LIN {X 0,Y 536.423,Z 174.915,A -85,B 0,C 180,E1 25056.548,E2 25056.548} C_VEL
LIN {X 0,Y 536.456,Z 174.916,A -85,B 0,C 180,E1 25053.19,E2 25053.19} C_VEL
LIN {X 0,Y 536.429,Z 174.979,A -85,B 0,C 180,E1 25052.229,E2 25052.229} C_VEL
LIN {X 0,Y 538.274,Z 182.198,A -85,B 0,C 180,E1 25051.657,E2 25051.657} C_VEL
LIN {X 0,Y 539.189,Z 215.155,A -85,B 0,C 180,E1 25049.25,E2 25049.25} C_VEL
LIN {X 0,Y 539.582,Z 245.329,A -85,B 0,C 180,E1 25046.881,E2 25046.881} C_VEL
LIN {X 0,Y 539.681,Z 277.796,A -85,B 0,C 180,E1 25044.228,E2 25044.228} C_VEL
LIN {X 0,Y 539.301,Z 312.385,A -85,B 0,C 180,E1 25041.251,E2 25041.251} C_VEL
LIN {X 0,Y 539.248,Z 319.143,A -85,B 0,C 180,E1 25040.702,E2 25040.702} C_VEL
LIN {X 0,Y 539.576,Z 325.813,A -85,B 0,C 180,E1 25040.595,E2 25040.595} C_VEL
LIN {X 0,Y 538.831,Z 486.501,A -85,B 0,C 180,E1 25038.368,E2 25038.368} C_VEL
LIN {X 0,Y 538.703,Z 503.712,A -85,B 0,C 180,E1 25037.931,E2 25037.931} C_VEL
LIN {X 0,Y 538.465,Z 519.532,A -85,B 0,C 180,E1 25037.339,E2 25037.339} C_VEL
LIN {X 0,Y 538.129,Z 535.901,A -85,B 0,C 180,E1 25036.514,E2 25036.514} C_VEL
LIN {X 0,Y 537.753,Z 551.043,A -85,B 0,C 180,E1 25035.53,E2 25035.53} C_VEL
LIN {X 0,Y 537.349,Z 564.974,A -85,B 0,C 180,E1 25034.383,E2 25034.383} C_VEL
LIN {X 0,Y 536.941,Z 578.306,A -85,B 0,C 180,E1 25033.021,E2 25033.021} C_VEL
LIN {X 0,Y 536.586,Z 589.487,A -85,B 0,C 180,E1 25031.609,E2 25031.609} C_VEL
LIN {X 0,Y 536.286,Z 599.811,A -85,B 0,C 180,E1 25029.985,E2 25029.985} C_VEL
LIN {X 0,Y 536.079,Z 608.451,A -85,B 0,C 180,E1 25028.257,E2 25028.257} C_VEL
LIN {X 0,Y 535.975,Z 615.684,A -85,B 0,C 180,E1 25026.426,E2 25026.426} C_VEL
LIN {X 0,Y 535.936,Z 620.745,A -85,B 0,C 180,E1 25024.708,E2 25024.708} C_VEL
LIN {X 0,Y 535.917,Z 624.48,A -85,B 0,C 180,E1 25022.78,E2 25022.78} C_VEL
LIN {X 0,Y 535.91,Z 626.276,A -85,B 0,C 180,E1 25020.855,E2 25020.855} C_VEL
LIN {X 0,Y 535.911,Z 626.268,A -85,B 0,C 180,E1 25019.038,E2 25019.038} C_VEL
LIN {X 0,Y 535.913,Z 624.459,A -85,B 0,C 180,E1 25017.112,E2 25017.112} C_VEL
LIN {X 0,Y 535.931,Z 620.697,A -85,B 0,C 180,E1 25015.184,E2 25015.184} C_VEL
LIN {X 0,Y 535.979,Z 615.244,A -85,B 0,C 180,E1 25013.358,E2 25013.358} C_VEL
LIN {X 0,Y 536.088,Z 607.834,A -85,B 0,C 180,E1 25011.527,E2 25011.527} C_VEL
LIN {X 0,Y 536.285,Z 599.404,A -85,B 0,C 180,E1 25009.872,E2 25009.872} C_VEL
LIN {X 0,Y 536.566,Z 589.166,A -85,B 0,C 180,E1 25008.28,E2 25008.28} C_VEL
LIN {X 0,Y 536.909,Z 577.887,A -85,B 0,C 180,E1 25006.868,E2 25006.868} C_VEL
LIN {X 0,Y 537.301,Z 565.067,A -85,B 0,C 180,E1 25005.56,E2 25005.56} C_VEL
LIN {X 0,Y 537.724,Z 550.492,A -85,B 0,C 180,E1 25004.358,E2 25004.358} C_VEL
LIN {X 0,Y 538.125,Z 535.397,A -85,B 0,C 180,E1 25003.373,E2 25003.373} C_VEL
LIN {X 0,Y 538.466,Z 519.15,A -85,B 0,C 180,E1 25002.549,E2 25002.549} C_VEL
LIN {X 0,Y 538.78,Z 502.032,A -85,B 0,C 180,E1 25001.907,E2 25001.907} C_VEL
LIN {X 0,Y 538.968,Z 484.452,A -85,B 0,C 180,E1 25001.468,E2 25001.468} C_VEL
LIN {X 0,Y 539.448,Z 388.201,A -85,B 0,C 180,E1 25000.124,E2 25000.124} C_VEL
LIN {X 0,Y 538.575,Z 380.596,A -85,B 0,C 180,E1 24999.986,E2 24999.986} C_VEL
LIN {X 0,Y 532.766,Z 360.688,A -85,B 0,C 180,E1 24999.487,E2 24999.487} C_VEL
LIN {X 0,Y 532.096,Z 354.154,A -85,B 0,C 180,E1 24999.367,E2 24999.367} C_VEL
LIN {X 0,Y 532.09,Z 321.506,A -85,B 0,C 180,E1 24998.896,E2 24998.896} C_VEL
LIN {X 0,Y 531.331,Z 316.809,A -85,B 0,C 180,E1 24998.79,E2 24998.79} C_VEL
LIN {X 0,Y 532.06,Z 279.719,A -85,B 0,C 180,E1 24995.408,E2 24995.408} C_VEL
LIN {X 0,Y 532.553,Z 244.005,A -85,B 0,C 180,E1 24992.165,E2 24992.165} C_VEL
LIN {X 0,Y 532.935,Z 207.634,A -85,B 0,C 180,E1 24988.87,E2 24988.87} C_VEL
LIN {X 0,Y 533.056,Z 191.079,A -85,B 0,C 180,E1 24987.373,E2 24987.373} C_VEL
LIN {X 0,Y 528.507,Z 175.902,A -85,B 0,C 180,E1 24985.715,E2 24985.715} C_VEL
LIN {X 0,Y 528.552,Z 176.121,A -85,B 0,C 180,E1 24984.625,E2 24984.625} C_VEL
LIN {X 0,Y 529.932,Z 179.548,A -85,B 0,C 180,E1 24984.453,E2 24984.453} C_VEL
LIN {X 0,Y 531.563,Z 181.867,A -85,B 0,C 180,E1 24984.281,E2 24984.281} C_VEL
LIN {X 0,Y 541.38,Z 197.994,A -85,B 0,C 180,E1 24983.233,E2 24983.233} C_VEL
LIN {X 0,Y 539.048,Z 419.645,A -85,B 0,C 180,E1 24979.896,E2 24979.896} C_VEL
LIN {X 0,Y 538.527,Z 464.266,A -85,B 0,C 180,E1 24979.196,E2 24979.196} C_VEL
LIN {X 0,Y 537.87,Z 485.766,A -85,B 0,C 180,E1 24978.667,E2 24978.667} C_VEL
LIN {X 0,Y 537.128,Z 506.444,A -85,B 0,C 180,E1 24977.965,E2 24977.965} C_VEL
LIN {X 0,Y 536.288,Z 525.333,A -85,B 0,C 180,E1 24977.154,E2 24977.154} C_VEL
LIN {X 0,Y 535.271,Z 545.952,A -85,B 0,C 180,E1 24976.063,E2 24976.063} C_VEL
LIN {X 0,Y 534.249,Z 564.528,A -85,B 0,C 180,E1 24974.875,E2 24974.875} C_VEL
LIN {X 0,Y 533.163,Z 583.881,A -85,B 0,C 180,E1 24973.418,E2 24973.418} C_VEL
LIN {X 0,Y 532.132,Z 600.696,A -85,B 0,C 180,E1 24971.92,E2 24971.92} C_VEL
LIN {X 0,Y 531.203,Z 617.415,A -85,B 0,C 180,E1 24970.212,E2 24970.212} C_VEL
LIN {X 0,Y 530.324,Z 633.077,A -85,B 0,C 180,E1 24968.337,E2 24968.337} C_VEL
LIN {X 0,Y 529.625,Z 646.645,A -85,B 0,C 180,E1 24966.463,E2 24966.463} C_VEL
LIN {X 0,Y 529.002,Z 660.204,A -85,B 0,C 180,E1 24964.281,E2 24964.281} C_VEL
LIN {X 0,Y 528.567,Z 671.632,A -85,B 0,C 180,E1 24962.111,E2 24962.111} C_VEL
LIN {X 0,Y 528.249,Z 682.226,A -85,B 0,C 180,E1 24959.681,E2 24959.681} C_VEL
LIN {X 0,Y 528.072,Z 689.894,A -85,B 0,C 180,E1 24957.516,E2 24957.516} C_VEL
LIN {X 0,Y 527.973,Z 696.696,A -85,B 0,C 180,E1 24955.101,E2 24955.101} C_VEL
LIN {X 0,Y 527.924,Z 701.372,A -85,B 0,C 180,E1 24952.846,E2 24952.846} C_VEL
LIN {X 0,Y 527.907,Z 704.615,A -85,B 0,C 180,E1 24950.511,E2 24950.511} C_VEL
LIN {X 0,Y 527.91,Z 706.258,A -85,B 0,C 180,E1 24948.097,E2 24948.097} C_VEL
LIN {X 0,Y 527.916,Z 706.289,A -85,B 0,C 180,E1 24945.94,E2 24945.94} C_VEL
LIN {X 0,Y 527.916,Z 704.805,A -85,B 0,C 180,E1 24943.583,E2 24943.583} C_VEL
LIN {X 0,Y 527.929,Z 701.693,A -85,B 0,C 180,E1 24941.249,E2 24941.249} C_VEL
LIN {X 0,Y 527.966,Z 697.241,A -85,B 0,C 180,E1 24939.044,E2 24939.044} C_VEL
LIN {X 0,Y 528.066,Z 690.659,A -85,B 0,C 180,E1 24936.633,E2 24936.633} C_VEL
LIN {X 0,Y 528.231,Z 683.073,A -85,B 0,C 180,E1 24934.451,E2 24934.451} C_VEL
LIN {X 0,Y 528.516,Z 673.375,A -85,B 0,C 180,E1 24932.169,E2 24932.169} C_VEL
LIN {X 0,Y 528.93,Z 662.117,A -85,B 0,C 180,E1 24929.97,E2 24929.97} C_VEL
LIN {X 0,Y 529.513,Z 649.292,A -85,B 0,C 180,E1 24927.836,E2 24927.836} C_VEL
LIN {X 0,Y 530.185,Z 635.52,A -85,B 0,C 180,E1 24925.891,E2 24925.891} C_VEL
LIN {X 0,Y 531.061,Z 619.631,A -85,B 0,C 180,E1 24923.948,E2 24923.948} C_VEL
LIN {X 0,Y 532.034,Z 602.565,A -85,B 0,C 180,E1 24922.169,E2 24922.169} C_VEL
LIN {X 0,Y 533.029,Z 585.876,A -85,B 0,C 180,E1 24920.662,E2 24920.662} C_VEL
LIN {X 0,Y 534.148,Z 566.313,A -85,B 0,C 180,E1 24919.157,E2 24919.157} C_VEL
LIN {X 0,Y 535.213,Z 547.196,A -85,B 0,C 180,E1 24917.923,E2 24917.923} C_VEL
LIN {X 0,Y 536.252,Z 526.209,A -85,B 0,C 180,E1 24916.797,E2 24916.797} C_VEL
LIN {X 0,Y 537.065,Z 507.68,A -85,B 0,C 180,E1 24915.994,E2 24915.994} C_VEL
LIN {X 0,Y 537.857,Z 487.102,A -85,B 0,C 180,E1 24915.28,E2 24915.28} C_VEL
LIN {X 0,Y 538.479,Z 465.319,A -85,B 0,C 180,E1 24914.736,E2 24914.736} C_VEL
LIN {X 0,Y 538.951,Z 430.041,A -85,B 0,C 180,E1 24914.169,E2 24914.169} C_VEL
LIN {X 0,Y 541.072,Z 221.448,A -85,B 0,C 180,E1 24911.031,E2 24911.031} C_VEL
LIN {X 0,Y 541.252,Z 197.496,A -85,B 0,C 180,E1 24910.659,E2 24910.659} C_VEL
LIN {X 0,Y 530.508,Z 180.267,A -85,B 0,C 180,E1 24909.507,E2 24909.507} C_VEL
LIN {X 0,Y 528.744,Z 177.007,A -85,B 0,C 180,E1 24909.3,E2 24909.3} C_VEL
LIN {X 0,Y 528.527,Z 175.903,A -85,B 0,C 180,E1 24909.234,E2 24909.234} C_VEL
LIN {X 0,Y 528.523,Z 175.903,A -85,B 0,C 180,E1 24905.763,E2 24905.763} C_VEL
LIN {X 0,Y 528.525,Z 175.902,A -85,B 0,C 180,E1 24902.265,E2 24902.265} C_VEL
LIN {X 0,Y 528.529,Z 175.899,A -85,B 0,C 180,E1 24898.77,E2 24898.77} C_VEL
LIN {X 0,Y 528.467,Z 175.902,A -85,B 0,C 180,E1 24895.417,E2 24895.417} C_VEL
LIN {X 0,Y 528.468,Z 175.898,A -85,B 0,C 180,E1 24892.056,E2 24892.056} C_VEL
LIN {X 0,Y 528.527,Z 175.892,A -85,B 0,C 180,E1 24888.827,E2 24888.827} C_VEL
LIN {X 0,Y 528.521,Z 175.894,A -85,B 0,C 180,E1 24885.343,E2 24885.343} C_VEL
LIN {X 0,Y 528.523,Z 175.899,A -85,B 0,C 180,E1 24881.898,E2 24881.898} C_VEL
LIN {X 0,Y 528.528,Z 175.901,A -85,B 0,C 180,E1 24878.446,E2 24878.446} C_VEL
LIN {X 0,Y 528.482,Z 175.901,A -85,B 0,C 180,E1 24875.111,E2 24875.111} C_VEL
LIN {X 0,Y 528.463,Z 175.896,A -85,B 0,C 180,E1 24871.735,E2 24871.735} C_VEL
LIN {X 0,Y 528.503,Z 175.896,A -85,B 0,C 180,E1 24868.351,E2 24868.351} C_VEL
LIN {X 0,Y 528.522,Z 175.899,A -85,B 0,C 180,E1 24864.953,E2 24864.953} C_VEL
LIN {X 0,Y 528.509,Z 175.902,A -85,B 0,C 180,E1 24861.442,E2 24861.442} C_VEL
LIN {X 0,Y 528.519,Z 175.894,A -85,B 0,C 180,E1 24858.075,E2 24858.075} C_VEL
LIN {X 0,Y 528.513,Z 175.903,A -85,B 0,C 180,E1 24854.685,E2 24854.685} C_VEL
LIN {X 0,Y 528.47,Z 175.904,A -85,B 0,C 180,E1 24851.348,E2 24851.348} C_VEL
LIN {X 0,Y 528.485,Z 175.897,A -85,B 0,C 180,E1 24847.939,E2 24847.939} C_VEL
LIN {X 0,Y 528.522,Z 175.889,A -85,B 0,C 180,E1 24844.558,E2 24844.558} C_VEL
LIN {X 0,Y 528.507,Z 175.898,A -85,B 0,C 180,E1 24841.193,E2 24841.193} C_VEL
LIN {X 0,Y 528.505,Z 175.903,A -85,B 0,C 180,E1 24837.723,E2 24837.723} C_VEL
LIN {X 0,Y 528.521,Z 175.901,A -85,B 0,C 180,E1 24834.319,E2 24834.319} C_VEL
LIN {X 0,Y 528.482,Z 175.9,A -85,B 0,C 180,E1 24830.966,E2 24830.966} C_VEL
LIN {X 0,Y 528.485,Z 175.898,A -85,B 0,C 180,E1 24827.656,E2 24827.656} C_VEL
LIN {X 0,Y 528.52,Z 175.896,A -85,B 0,C 180,E1 24824.305,E2 24824.305} C_VEL
LIN {X 0,Y 528.508,Z 175.901,A -85,B 0,C 180,E1 24820.896,E2 24820.896} C_VEL
LIN {X 0,Y 528.498,Z 175.904,A -85,B 0,C 180,E1 24817.405,E2 24817.405} C_VEL
LIN {X 0,Y 528.514,Z 175.9,A -85,B 0,C 180,E1 24814.087,E2 24814.087} C_VEL
LIN {X 0,Y 528.498,Z 175.899,A -85,B 0,C 180,E1 24810.66,E2 24810.66} C_VEL
LIN {X 0,Y 528.551,Z 176.084,A -85,B 0,C 180,E1 24808.369,E2 24808.369} C_VEL
LIN {X 0,Y 529.95,Z 179.609,A -85,B 0,C 180,E1 24807.901,E2 24807.901} C_VEL
LIN {X 0,Y 536.933,Z 193.998,A -85,B 0,C 180,E1 24805.909,E2 24805.909} C_VEL
LIN {X 0,Y 542.938,Z 206.96,A -85,B 0,C 180,E1 24804.219,E2 24804.219} C_VEL
LIN {X 0,Y 541.161,Z 250.131,A -85,B 0,C 180,E1 24800.896,E2 24800.896} C_VEL
LIN {X 0,Y 540.404,Z 281.034,A -85,B 0,C 180,E1 24798.533,E2 24798.533} C_VEL
LIN {X 0,Y 541.806,Z 294.589,A -85,B 0,C 180,E1 24797.37,E2 24797.37} C_VEL
LIN {X 0,Y 544.881,Z 306.361,A -85,B 0,C 180,E1 24796.228,E2 24796.228} C_VEL
LIN {X 0,Y 549.168,Z 315.707,A -85,B 0,C 180,E1 24795.203,E2 24795.203} C_VEL
LIN {X 0,Y 555.008,Z 323.69,A -85,B 0,C 180,E1 24794.193,E2 24794.193} C_VEL
LIN {X 0,Y 561.764,Z 329.796,A -85,B 0,C 180,E1 24793.285,E2 24793.285} C_VEL
LIN {X 0,Y 569.988,Z 334.684,A -85,B 0,C 180,E1 24792.396,E2 24792.396} C_VEL
LIN {X 0,Y 574.04,Z 336.198,A -85,B 0,C 180,E1 24791.949,E2 24791.949} C_VEL
LIN {X 0,Y 577.589,Z 336.609,A -85,B 0,C 180,E1 24791.397,E2 24791.397} C_VEL
LIN {X 0,Y 580.095,Z 335.749,A -85,B 0,C 180,E1 24790.787,E2 24790.787} C_VEL
LIN {X 0,Y 581.221,Z 333.782,A -85,B 0,C 180,E1 24790.173,E2 24790.173} C_VEL
LIN {X 0,Y 580.918,Z 330.792,A -85,B 0,C 180,E1 24789.588,E2 24789.588} C_VEL
LIN {X 0,Y 579.132,Z 326.906,A -85,B 0,C 180,E1 24789.062,E2 24789.062} C_VEL
LIN {X 0,Y 574.303,Z 319.616,A -85,B 0,C 180,E1 24788.412,E2 24788.412} C_VEL
LIN {X 0,Y 568.986,Z 309.485,A -85,B 0,C 180,E1 24787.732,E2 24787.732} C_VEL
LIN {X 0,Y 564.615,Z 298.029,A -85,B 0,C 180,E1 24787.155,E2 24787.155} C_VEL
LIN {X 0,Y 561.237,Z 285.291,A -85,B 0,C 180,E1 24786.697,E2 24786.697} C_VEL
LIN {X 0,Y 560.435,Z 281.641,A -85,B 0,C 180,E1 24786.587,E2 24786.587} C_VEL
LIN {X 0,Y 556.42,Z 319.177,A -85,B 0,C 180,E1 24786.027,E2 24786.027} C_VEL
LIN {X 0,Y 553.604,Z 338.038,A -85,B 0,C 180,E1 24785.624,E2 24785.624} C_VEL
LIN {X 0,Y 551.79,Z 345.175,A -85,B 0,C 180,E1 24785.36,E2 24785.36} C_VEL
LIN {X 0,Y 551.411,Z 347.117,A -85,B 0,C 180,E1 24785.305,E2 24785.305} C_VEL
LIN {X 0,Y 547.128,Z 398.954,A -85,B 0,C 180,E1 24784.666,E2 24784.666} C_VEL
LIN {X 0,Y 544.19,Z 425.471,A -85,B 0,C 180,E1 24784.245,E2 24784.245} C_VEL
LIN {X 0,Y 541.514,Z 438.292,A -85,B 0,C 180,E1 24783.923,E2 24783.923} C_VEL
LIN {X 0,Y 539.664,Z 444.325,A -85,B 0,C 180,E1 24783.64,E2 24783.64} C_VEL
LIN {X 0,Y 539.454,Z 449.477,A -85,B 0,C 180,E1 24783.539,E2 24783.539} C_VEL
LIN {X 0,Y 538.548,Z 532.883,A -85,B 0,C 180,E1 24782.268,E2 24782.268} C_VEL
LIN {X 0,Y 537.912,Z 554.763,A -85,B 0,C 180,E1 24781.742,E2 24781.742} C_VEL
LIN {X 0,Y 537.113,Z 577.319,A -85,B 0,C 180,E1 24780.978,E2 24780.978} C_VEL
LIN {X 0,Y 536.158,Z 598.433,A -85,B 0,C 180,E1 24780.053,E2 24780.053} C_VEL
LIN {X 0,Y 535.138,Z 618.797,A -85,B 0,C 180,E1 24778.942,E2 24778.942} C_VEL
LIN {X 0,Y 534.006,Z 638.991,A -85,B 0,C 180,E1 24777.607,E2 24777.607} C_VEL
LIN {X 0,Y 532.849,Z 658.823,A -85,B 0,C 180,E1 24776.045,E2 24776.045} C_VEL
LIN {X 0,Y 531.812,Z 676.835,A -85,B 0,C 180,E1 24774.373,E2 24774.373} C_VEL
LIN {X 0,Y 530.823,Z 694.223,A -85,B 0,C 180,E1 24772.48,E2 24772.48} C_VEL
LIN {X 0,Y 529.961,Z 710.289,A -85,B 0,C 180,E1 24770.428,E2 24770.428} C_VEL
LIN {X 0,Y 529.261,Z 724.605,A -85,B 0,C 180,E1 24768.276,E2 24768.276} C_VEL
LIN {X 0,Y 528.723,Z 737.275,A -85,B 0,C 180,E1 24766.027,E2 24766.027} C_VEL
LIN {X 0,Y 528.359,Z 748.319,A -85,B 0,C 180,E1 24763.683,E2 24763.683} C_VEL
LIN {X 0,Y 528.13,Z 757.313,A -85,B 0,C 180,E1 24761.355,E2 24761.355} C_VEL
LIN {X 0,Y 528.003,Z 764.399,A -85,B 0,C 180,E1 24759.043,E2 24759.043} C_VEL
LIN {X 0,Y 527.934,Z 770.012,A -85,B 0,C 180,E1 24756.634,E2 24756.634} C_VEL
LIN {X 0,Y 527.915,Z 773.739,A -85,B 0,C 180,E1 24754.345,E2 24754.345} C_VEL
LIN {X 0,Y 527.91,Z 775.902,A -85,B 0,C 180,E1 24751.954,E2 24751.954} C_VEL
LIN {X 0,Y 527.898,Z 776.445,A -85,B 0,C 180,E1 24749.566,E2 24749.566} C_VEL
LIN {X 0,Y 527.913,Z 775.33,A -85,B 0,C 180,E1 24747.177,E2 24747.177} C_VEL
LIN {X 0,Y 527.924,Z 772.489,A -85,B 0,C 180,E1 24744.784,E2 24744.784} C_VEL
LIN {X 0,Y 527.954,Z 767.939,A -85,B 0,C 180,E1 24742.382,E2 24742.382} C_VEL
LIN {X 0,Y 528.032,Z 761.923,A -85,B 0,C 180,E1 24740.077,E2 24740.077} C_VEL
LIN {X 0,Y 528.201,Z 754.099,A -85,B 0,C 180,E1 24737.76,E2 24737.76} C_VEL
LIN {X 0,Y 528.486,Z 744.355,A -85,B 0,C 180,E1 24735.426,E2 24735.426} C_VEL
LIN {X 0,Y 528.903,Z 733.12,A -85,B 0,C 180,E1 24733.187,E2 24733.187} C_VEL
LIN {X 0,Y 529.499,Z 719.628,A -85,B 0,C 180,E1 24730.933,E2 24730.933} C_VEL
LIN {X 0,Y 530.264,Z 704.345,A -85,B 0,C 180,E1 24728.775,E2 24728.775} C_VEL
LIN {X 0,Y 531.183,Z 687.693,A -85,B 0,C 180,E1 24726.775,E2 24726.775} C_VEL
LIN {X 0,Y 532.217,Z 669.663,A -85,B 0,C 180,E1 24724.929,E2 24724.929} C_VEL
LIN {X 0,Y 533.303,Z 651.138,A -85,B 0,C 180,E1 24723.319,E2 24723.319} C_VEL
LIN {X 0,Y 534.442,Z 631.515,A -85,B 0,C 180,E1 24721.871,E2 24721.871} C_VEL
LIN {X 0,Y 535.478,Z 611.858,A -85,B 0,C 180,E1 24720.656,E2 24720.656} C_VEL
LIN {X 0,Y 536.518,Z 591.146,A -85,B 0,C 180,E1 24719.604,E2 24719.604} C_VEL
LIN {X 0,Y 537.396,Z 569.684,A -85,B 0,C 180,E1 24718.736,E2 24718.736} C_VEL
LIN {X 0,Y 538.157,Z 547.837,A -85,B 0,C 180,E1 24718.07,E2 24718.07} C_VEL
LIN {X 0,Y 538.658,Z 525.76,A -85,B 0,C 180,E1 24717.604,E2 24717.604} C_VEL
LIN {X 0,Y 539.775,Z 430.01,A -85,B 0,C 180,E1 24716.152,E2 24716.152} C_VEL
LIN {X 0,Y 542.023,Z 420.357,A -85,B 0,C 180,E1 24715.786,E2 24715.786} C_VEL
LIN {X 0,Y 545.471,Z 402.426,A -85,B 0,C 180,E1 24715.391,E2 24715.391} C_VEL
LIN {X 0,Y 548.926,Z 377.608,A -85,B 0,C 180,E1 24715.046,E2 24715.046} C_VEL
LIN {X 0,Y 551.647,Z 345.727,A -85,B 0,C 180,E1 24714.661,E2 24714.661} C_VEL
LIN {X 0,Y 553.46,Z 338.838,A -85,B 0,C 180,E1 24714.397,E2 24714.397} C_VEL
LIN {X 0,Y 556.257,Z 320.33,A -85,B 0,C 180,E1 24713.996,E2 24713.996} C_VEL
LIN {X 0,Y 560.306,Z 282.948,A -85,B 0,C 180,E1 24713.43,E2 24713.43} C_VEL
LIN {X 0,Y 563.751,Z 243.723,A -85,B 0,C 180,E1 24712.961,E2 24712.961} C_VEL
LIN {X 0,Y 566.397,Z 236.791,A -85,B 0,C 180,E1 24712.608,E2 24712.608} C_VEL
LIN {X 0,Y 570.674,Z 224.702,A -85,B 0,C 180,E1 24712.05,E2 24712.05} C_VEL
LIN {X 0,Y 578.916,Z 233.762,A -85,B 0,C 180,E1 24711.016,E2 24711.016} C_VEL
LIN {X 0,Y 584.234,Z 238.146,A -85,B 0,C 180,E1 24710.331,E2 24710.331} C_VEL
LIN {X 0,Y 586.631,Z 240.449,A -85,B 0,C 180,E1 24709.761,E2 24709.761} C_VEL
LIN {X 0,Y 587.526,Z 242.015,A -85,B 0,C 180,E1 24709.123,E2 24709.123} C_VEL
LIN {X 0,Y 586.921,Z 242.678,A -85,B 0,C 180,E1 24708.495,E2 24708.495} C_VEL
LIN {X 0,Y 584.777,Z 243.17,A -85,B 0,C 180,E1 24707.907,E2 24707.907} C_VEL
LIN {X 0,Y 581.547,Z 242.701,A -85,B 0,C 180,E1 24707.38,E2 24707.38} C_VEL
LIN {X 0,Y 576.792,Z 240.967,A -85,B 0,C 180,E1 24706.869,E2 24706.869} C_VEL
LIN {X 0,Y 568.313,Z 236.051,A -85,B 0,C 180,E1 24706.019,E2 24706.019} C_VEL
LIN {X 0,Y 557.073,Z 227.173,A -85,B 0,C 180,E1 24704.714,E2 24704.714} C_VEL
LIN {X 0,Y 550.573,Z 219.37,A -85,B 0,C 180,E1 24703.781,E2 24703.781} C_VEL
LIN {X 0,Y 543.109,Z 205.081,A -85,B 0,C 180,E1 24702.361,E2 24702.361} C_VEL
LIN {X 0,Y 534.69,Z 188.296,A -85,B 0,C 180,E1 24700.598,E2 24700.598} C_VEL
LIN {X 0,Y 530.631,Z 180.384,A -85,B 0,C 180,E1 24699.7,E2 24699.7} C_VEL
LIN {X 0,Y 528.79,Z 177.165,A -85,B 0,C 180,E1 24699.303,E2 24699.303} C_VEL
LIN {X 0,Y 528.526,Z 175.9,A -85,B 0,C 180,E1 24699.187,E2 24699.187} C_VEL
LIN {X 0,Y 528.518,Z 175.894,A -85,B 0,C 180,E1 24695.748,E2 24695.748} C_VEL
LIN {X 0,Y 528.503,Z 176.088,A -85,B 0,C 180,E1 24692.499,E2 24692.499} C_VEL
LIN {X 0,Y 530.725,Z 184.55,A -85,B 0,C 180,E1 24691.825,E2 24691.825} C_VEL
LIN {X 0,Y 531.673,Z 218.661,A -85,B 0,C 180,E1 24689.333,E2 24689.333} C_VEL
LIN {X 0,Y 532.08,Z 248.562,A -85,B 0,C 180,E1 24686.988,E2 24686.988} C_VEL
LIN {X 0,Y 532.161,Z 277.939,A -85,B 0,C 180,E1 24684.581,E2 24684.581} C_VEL
LIN {X 0,Y 531.869,Z 311.423,A -85,B 0,C 180,E1 24681.736,E2 24681.736} C_VEL
LIN {X 0,Y 531.754,Z 320.791,A -85,B 0,C 180,E1 24680.944,E2 24680.944} C_VEL
LIN {X 0,Y 531.844,Z 345.536,A -85,B 0,C 180,E1 24680.577,E2 24680.577} C_VEL
LIN {X 0,Y 531.11,Z 488.372,A -85,B 0,C 180,E1 24678.56,E2 24678.56} C_VEL
LIN {X 0,Y 530.993,Z 505.555,A -85,B 0,C 180,E1 24678.115,E2 24678.115} C_VEL
LIN {X 0,Y 530.746,Z 521.979,A -85,B 0,C 180,E1 24677.486,E2 24677.486} C_VEL
LIN {X 0,Y 530.41,Z 538.189,A -85,B 0,C 180,E1 24676.65,E2 24676.65} C_VEL
LIN {X 0,Y 530.023,Z 553.212,A -85,B 0,C 180,E1 24675.65,E2 24675.65} C_VEL
LIN {X 0,Y 529.601,Z 567.045,A -85,B 0,C 180,E1 24674.486,E2 24674.486} C_VEL
LIN {X 0,Y 529.201,Z 579.327,A -85,B 0,C 180,E1 24673.215,E2 24673.215} C_VEL
LIN {X 0,Y 528.823,Z 590.633,A -85,B 0,C 180,E1 24671.782,E2 24671.782} C_VEL
LIN {X 0,Y 528.513,Z 600.439,A -85,B 0,C 180,E1 24670.243,E2 24670.243} C_VEL
LIN {X 0,Y 528.282,Z 608.779,A -85,B 0,C 180,E1 24668.599,E2 24668.599} C_VEL
LIN {X 0,Y 528.11,Z 616.086,A -85,B 0,C 180,E1 24666.741,E2 24666.741} C_VEL
LIN {X 0,Y 528.005,Z 621.378,A -85,B 0,C 180,E1 24664.888,E2 24664.888} C_VEL
LIN {X 0,Y 527.953,Z 625.014,A -85,B 0,C 180,E1 24662.931,E2 24662.931} C_VEL
LIN {X 0,Y 527.934,Z 626.814,A -85,B 0,C 180,E1 24660.976,E2 24660.976} C_VEL
LIN {X 0,Y 527.933,Z 626.896,A -85,B 0,C 180,E1 24659.131,E2 24659.131} C_VEL
LIN {X 0,Y 527.943,Z 625.236,A -85,B 0,C 180,E1 24657.177,E2 24657.177} C_VEL
LIN {X 0,Y 527.981,Z 621.708,A -85,B 0,C 180,E1 24655.22,E2 24655.22} C_VEL
LIN {X 0,Y 528.068,Z 616.563,A -85,B 0,C 180,E1 24653.367,E2 24653.367} C_VEL
LIN {X 0,Y 528.214,Z 609.907,A -85,B 0,C 180,E1 24651.619,E2 24651.619} C_VEL
LIN {X 0,Y 528.43,Z 601.211,A -85,B 0,C 180,E1 24649.865,E2 24649.865} C_VEL
LIN {X 0,Y 528.741,Z 590.86,A -85,B 0,C 180,E1 24648.215,E2 24648.215} C_VEL
LIN {X 0,Y 529.107,Z 579.659,A -85,B 0,C 180,E1 24646.782,E2 24646.782} C_VEL
LIN {X 0,Y 529.521,Z 566.914,A -85,B 0,C 180,E1 24645.455,E2 24645.455} C_VEL
LIN {X 0,Y 529.953,Z 553.191,A -85,B 0,C 180,E1 24644.291,E2 24644.291} C_VEL
LIN {X 0,Y 530.387,Z 538.16,A -85,B 0,C 180,E1 24643.268,E2 24643.268} C_VEL
LIN {X 0,Y 530.733,Z 522.867,A -85,B 0,C 180,E1 24642.456,E2 24642.456} C_VEL
LIN {X 0,Y 531.068,Z 505.572,A -85,B 0,C 180,E1 24641.769,E2 24641.769} C_VEL
LIN {X 0,Y 531.288,Z 488.117,A -85,B 0,C 180,E1 24641.291,E2 24641.291} C_VEL
LIN {X 0,Y 531.434,Z 457.702,A -85,B 0,C 180,E1 24640.83,E2 24640.83} C_VEL
LIN {X 0,Y 532.096,Z 354.154,A -85,B 0,C 180,E1 24639.367,E2 24639.367} C_VEL
LIN {X 0,Y 531.148,Z 345.477,A -85,B 0,C 180,E1 24639.206,E2 24639.206} C_VEL
LIN {X 0,Y 524.384,Z 321.29,A -85,B 0,C 180,E1 24638.586,E2 24638.586} C_VEL
LIN {X 0,Y 524.194,Z 320.205,A -85,B 0,C 180,E1 24638.562,E2 24638.562} C_VEL
LIN {X 0,Y 523.811,Z 317.807,A -85,B 0,C 180,E1 24638.5,E2 24638.5} C_VEL
LIN {X 0,Y 524.559,Z 280.427,A -85,B 0,C 180,E1 24635.086,E2 24635.086} C_VEL
LIN {X 0,Y 525.105,Z 244.67,A -85,B 0,C 180,E1 24631.821,E2 24631.821} C_VEL
LIN {X 0,Y 525.533,Z 209.156,A -85,B 0,C 180,E1 24628.58,E2 24628.58} C_VEL
LIN {X 0,Y 525.615,Z 193.609,A -85,B 0,C 180,E1 24627.17,E2 24627.17} C_VEL
LIN {X 0,Y 520.585,Z 176.89,A -85,B 0,C 180,E1 24625.32,E2 24625.32} C_VEL
LIN {X 0,Y 520.713,Z 177.631,A -85,B 0,C 180,E1 24625.262,E2 24625.262} C_VEL
LIN {X 0,Y 522.321,Z 180.956,A -85,B 0,C 180,E1 24625.068,E2 24625.068} C_VEL
LIN {X 0,Y 523.757,Z 183.026,A -85,B 0,C 180,E1 24624.91,E2 24624.91} C_VEL
LIN {X 0,Y 534.892,Z 201.052,A -85,B 0,C 180,E1 24623.694,E2 24623.694} C_VEL
LIN {X 0,Y 532.311,Z 422.026,A -85,B 0,C 180,E1 24620.329,E2 24620.329} C_VEL
LIN {X 0,Y 531.746,Z 464.567,A -85,B 0,C 180,E1 24619.651,E2 24619.651} C_VEL
LIN {X 0,Y 531.028,Z 486.095,A -85,B 0,C 180,E1 24619.114,E2 24619.114} C_VEL
LIN {X 0,Y 530.161,Z 507.669,A -85,B 0,C 180,E1 24618.367,E2 24618.367} C_VEL
LIN {X 0,Y 529.171,Z 528.059,A -85,B 0,C 180,E1 24617.468,E2 24617.468} C_VEL
LIN {X 0,Y 528.001,Z 548.535,A -85,B 0,C 180,E1 24616.335,E2 24616.335} C_VEL
LIN {X 0,Y 526.839,Z 567.797,A -85,B 0,C 180,E1 24615.064,E2 24615.064} C_VEL
LIN {X 0,Y 525.574,Z 587.24,A -85,B 0,C 180,E1 24613.526,E2 24613.526} C_VEL
LIN {X 0,Y 524.525,Z 603.061,A -85,B 0,C 180,E1 24612.07,E2 24612.07} C_VEL
LIN {X 0,Y 523.397,Z 620.891,A -85,B 0,C 180,E1 24610.17,E2 24610.17} C_VEL
LIN {X 0,Y 522.422,Z 636.731,A -85,B 0,C 180,E1 24608.184,E2 24608.184} C_VEL
LIN {X 0,Y 521.595,Z 651.536,A -85,B 0,C 180,E1 24606.006,E2 24606.006} C_VEL
LIN {X 0,Y 521.036,Z 663.209,A -85,B 0,C 180,E1 24604.003,E2 24604.003} C_VEL
LIN {X 0,Y 520.55,Z 674.961,A -85,B 0,C 180,E1 24601.626,E2 24601.626} C_VEL
LIN {X 0,Y 520.24,Z 684.219,A -85,B 0,C 180,E1 24599.347,E2 24599.347} C_VEL
LIN {X 0,Y 520.057,Z 692.062,A -85,B 0,C 180,E1 24596.984,E2 24596.984} C_VEL
LIN {X 0,Y 519.963,Z 697.972,A -85,B 0,C 180,E1 24594.663,E2 24594.663} C_VEL
LIN {X 0,Y 519.93,Z 702.48,A -85,B 0,C 180,E1 24592.262,E2 24592.262} C_VEL
LIN {X 0,Y 519.904,Z 705.326,A -85,B 0,C 180,E1 24589.784,E2 24589.784} C_VEL
LIN {X 0,Y 519.902,Z 706.383,A -85,B 0,C 180,E1 24587.574,E2 24587.574} C_VEL
LIN {X 0,Y 519.912,Z 705.985,A -85,B 0,C 180,E1 24585.111,E2 24585.111} C_VEL
LIN {X 0,Y 519.909,Z 703.983,A -85,B 0,C 180,E1 24582.777,E2 24582.777} C_VEL
LIN {X 0,Y 519.927,Z 700.587,A -85,B 0,C 180,E1 24580.527,E2 24580.527} C_VEL
LIN {X 0,Y 519.996,Z 695.163,A -85,B 0,C 180,E1 24578.069,E2 24578.069} C_VEL
LIN {X 0,Y 520.117,Z 689.023,A -85,B 0,C 180,E1 24575.959,E2 24575.959} C_VEL
LIN {X 0,Y 520.356,Z 680.682,A -85,B 0,C 180,E1 24573.636,E2 24573.636} C_VEL
LIN {X 0,Y 520.698,Z 670.974,A -85,B 0,C 180,E1 24571.431,E2 24571.431} C_VEL
LIN {X 0,Y 521.165,Z 660.1,A -85,B 0,C 180,E1 24569.341,E2 24569.341} C_VEL
LIN {X 0,Y 521.896,Z 645.906,A -85,B 0,C 180,E1 24567.035,E2 24567.035} C_VEL
LIN {X 0,Y 522.671,Z 632.541,A -85,B 0,C 180,E1 24565.172,E2 24565.172} C_VEL
LIN {X 0,Y 523.732,Z 615.628,A -85,B 0,C 180,E1 24563.147,E2 24563.147} C_VEL
LIN {X 0,Y 524.717,Z 600.202,A -85,B 0,C 180,E1 24561.563,E2 24561.563} C_VEL
LIN {X 0,Y 525.934,Z 581.849,A -85,B 0,C 180,E1 24559.927,E2 24559.927} C_VEL
LIN {X 0,Y 527.068,Z 564.017,A -85,B 0,C 180,E1 24558.584,E2 24558.584} C_VEL
LIN {X 0,Y 528.21,Z 545.198,A -85,B 0,C 180,E1 24557.371,E2 24557.371} C_VEL
LIN {X 0,Y 529.323,Z 524.722,A -85,B 0,C 180,E1 24556.287,E2 24556.287} C_VEL
LIN {X 0,Y 530.199,Z 506.582,A -85,B 0,C 180,E1 24555.502,E2 24555.502} C_VEL
LIN {X 0,Y 531.054,Z 485.836,A -85,B 0,C 180,E1 24554.787,E2 24554.787} C_VEL
LIN {X 0,Y 531.757,Z 463.918,A -85,B 0,C 180,E1 24554.245,E2 24554.245} C_VEL
LIN {X 0,Y 532.44,Z 409.987,A -85,B 0,C 180,E1 24553.399,E2 24553.399} C_VEL
LIN {X 0,Y 534.845,Z 200.897,A -85,B 0,C 180,E1 24550.209,E2 24550.209} C_VEL
LIN {X 0,Y 524.951,Z 184.974,A -85,B 0,C 180,E1 24549.107,E2 24549.107} C_VEL
LIN {X 0,Y 522.762,Z 181.449,A -85,B 0,C 180,E1 24548.854,E2 24548.854} C_VEL
LIN {X 0,Y 520.877,Z 178.302,A -85,B 0,C 180,E1 24548.629,E2 24548.629} C_VEL
LIN {X 0,Y 520.566,Z 176.891,A -85,B 0,C 180,E1 24548.567,E2 24548.567} C_VEL
LIN {X 0,Y 520.582,Z 176.891,A -85,B 0,C 180,E1 24545.126,E2 24545.126} C_VEL
LIN {X 0,Y 520.563,Z 176.887,A -85,B 0,C 180,E1 24541.606,E2 24541.606} C_VEL
LIN {X 0,Y 520.568,Z 176.886,A -85,B 0,C 180,E1 24538.246,E2 24538.246} C_VEL
LIN {X 0,Y 520.572,Z 176.885,A -85,B 0,C 180,E1 24534.816,E2 24534.816} C_VEL
LIN {X 0,Y 520.553,Z 176.886,A -85,B 0,C 180,E1 24531.373,E2 24531.373} C_VEL
LIN {X 0,Y 520.554,Z 176.883,A -85,B 0,C 180,E1 24528.017,E2 24528.017} C_VEL
LIN {X 0,Y 520.578,Z 176.879,A -85,B 0,C 180,E1 24524.511,E2 24524.511} C_VEL
LIN {X 0,Y 520.568,Z 176.882,A -85,B 0,C 180,E1 24521.063,E2 24521.063} C_VEL
LIN {X 0,Y 520.543,Z 176.889,A -85,B 0,C 180,E1 24517.649,E2 24517.649} C_VEL
LIN {X 0,Y 520.544,Z 176.894,A -85,B 0,C 180,E1 24514.25,E2 24514.25} C_VEL
LIN {X 0,Y 520.589,Z 176.886,A -85,B 0,C 180,E1 24510.849,E2 24510.849} C_VEL
LIN {X 0,Y 520.57,Z 176.883,A -85,B 0,C 180,E1 24507.45,E2 24507.45} C_VEL
LIN {X 0,Y 520.573,Z 176.89,A -85,B 0,C 180,E1 24504.029,E2 24504.029} C_VEL
LIN {X 0,Y 520.586,Z 176.887,A -85,B 0,C 180,E1 24500.578,E2 24500.578} C_VEL
LIN {X 0,Y 520.545,Z 176.887,A -85,B 0,C 180,E1 24497.206,E2 24497.206} C_VEL
LIN {X 0,Y 520.522,Z 176.885,A -85,B 0,C 180,E1 24493.78,E2 24493.78} C_VEL
LIN {X 0,Y 520.568,Z 176.889,A -85,B 0,C 180,E1 24490.402,E2 24490.402} C_VEL
LIN {X 0,Y 520.59,Z 176.891,A -85,B 0,C 180,E1 24486.95,E2 24486.95} C_VEL
LIN {X 0,Y 520.581,Z 176.884,A -85,B 0,C 180,E1 24483.414,E2 24483.414} C_VEL
LIN {X 0,Y 520.588,Z 176.882,A -85,B 0,C 180,E1 24479.89,E2 24479.89} C_VEL
LIN {X 0,Y 520.586,Z 176.886,A -85,B 0,C 180,E1 24476.366,E2 24476.366} C_VEL
LIN {X 0,Y 520.527,Z 176.895,A -85,B 0,C 180,E1 24473.05,E2 24473.05} C_VEL
LIN {X 0,Y 520.534,Z 176.893,A -85,B 0,C 180,E1 24469.566,E2 24469.566} C_VEL
LIN {X 0,Y 520.567,Z 176.889,A -85,B 0,C 180,E1 24466.109,E2 24466.109} C_VEL
LIN {X 0,Y 520.581,Z 176.887,A -85,B 0,C 180,E1 24462.663,E2 24462.663} C_VEL
LIN {X 0,Y 520.562,Z 176.885,A -85,B 0,C 180,E1 24459.186,E2 24459.186} C_VEL
LIN {X 0,Y 520.57,Z 176.886,A -85,B 0,C 180,E1 24455.829,E2 24455.829} C_VEL
LIN {X 0,Y 520.57,Z 176.89,A -85,B 0,C 180,E1 24452.427,E2 24452.427} C_VEL
LIN {X 0,Y 520.539,Z 176.915,A -85,B 0,C 180,E1 24449.216,E2 24449.216} C_VEL
LIN {X 0,Y 521.966,Z 180.496,A -85,B 0,C 180,E1 24448.727,E2 24448.727} C_VEL
LIN {X 0,Y 523.024,Z 182.634,A -85,B 0,C 180,E1 24448.413,E2 24448.413} C_VEL
LIN {X 0,Y 530.735,Z 198.422,A -85,B 0,C 180,E1 24446.182,E2 24446.182} C_VEL
LIN {X 0,Y 536.458,Z 210.894,A -85,B 0,C 180,E1 24444.537,E2 24444.537} C_VEL
LIN {X 0,Y 534.514,Z 253.973,A -85,B 0,C 180,E1 24441.197,E2 24441.197} C_VEL
LIN {X 0,Y 533.681,Z 283.061,A -85,B 0,C 180,E1 24438.954,E2 24438.954} C_VEL
LIN {X 0,Y 535.005,Z 297.391,A -85,B 0,C 180,E1 24437.717,E2 24437.717} C_VEL
LIN {X 0,Y 538.123,Z 309.918,A -85,B 0,C 180,E1 24436.496,E2 24436.496} C_VEL
LIN {X 0,Y 542.519,Z 319.88,A -85,B 0,C 180,E1 24435.398,E2 24435.398} C_VEL
LIN {X 0,Y 548.238,Z 328.088,A -85,B 0,C 180,E1 24434.364,E2 24434.364} C_VEL
LIN {X 0,Y 554.843,Z 334.508,A -85,B 0,C 180,E1 24433.429,E2 24433.429} C_VEL
LIN {X 0,Y 562.878,Z 339.814,A -85,B 0,C 180,E1 24432.509,E2 24432.509} C_VEL
LIN {X 0,Y 569.997,Z 342.935,A -85,B 0,C 180,E1 24431.797,E2 24431.797} C_VEL
LIN {X 0,Y 573.672,Z 343.626,A -85,B 0,C 180,E1 24431.306,E2 24431.306} C_VEL
LIN {X 0,Y 576.605,Z 343.191,A -85,B 0,C 180,E1 24430.732,E2 24430.732} C_VEL
LIN {X 0,Y 578.263,Z 341.767,A -85,B 0,C 180,E1 24430.16,E2 24430.16} C_VEL
LIN {X 0,Y 578.675,Z 339.201,A -85,B 0,C 180,E1 24429.547,E2 24429.547} C_VEL
LIN {X 0,Y 577.541,Z 335.649,A -85,B 0,C 180,E1 24428.97,E2 24428.97} C_VEL
LIN {X 0,Y 574.924,Z 331.398,A -85,B 0,C 180,E1 24428.49,E2 24428.49} C_VEL
LIN {X 0,Y 568.832,Z 321.855,A -85,B 0,C 180,E1 24427.712,E2 24427.712} C_VEL
LIN {X 0,Y 563.599,Z 310.773,A -85,B 0,C 180,E1 24427.018,E2 24427.018} C_VEL
LIN {X 0,Y 562.547,Z 308.398,A -85,B 0,C 180,E1 24426.876,E2 24426.876} C_VEL
LIN {X 0,Y 559.115,Z 334.566,A -85,B 0,C 180,E1 24426.405,E2 24426.405} C_VEL
LIN {X 0,Y 556.788,Z 346.134,A -85,B 0,C 180,E1 24426.079,E2 24426.079} C_VEL
LIN {X 0,Y 555.925,Z 349.61,A -85,B 0,C 180,E1 24425.956,E2 24425.956} C_VEL
LIN {X 0,Y 551.523,Z 401.233,A -85,B 0,C 180,E1 24425.33,E2 24425.33} C_VEL
LIN {X 0,Y 548.301,Z 420.968,A -85,B 0,C 180,E1 24425.103,E2 24425.103} C_VEL
LIN {X 0,Y 544.402,Z 436.109,A -85,B 0,C 180,E1 24424.842,E2 24424.842} C_VEL
LIN {X 0,Y 541.4,Z 445.795,A -85,B 0,C 180,E1 24424.515,E2 24424.515} C_VEL
LIN {X 0,Y 540.488,Z 448.656,A -85,B 0,C 180,E1 24424.401,E2 24424.401} C_VEL
LIN {X 0,Y 536.627,Z 460.712,A -85,B 0,C 180,E1 24424.181,E2 24424.181} C_VEL
LIN {X 0,Y 533.455,Z 470.211,A -85,B 0,C 180,E1 24423.826,E2 24423.826} C_VEL
LIN {X 0,Y 532.508,Z 473.779,A -85,B 0,C 180,E1 24423.649,E2 24423.649} C_VEL
LIN {X 0,Y 531.769,Z 533.222,A -85,B 0,C 180,E1 24422.722,E2 24422.722} C_VEL
LIN {X 0,Y 531.076,Z 555.006,A -85,B 0,C 180,E1 24422.191,E2 24422.191} C_VEL
LIN {X 0,Y 530.198,Z 577.313,A -85,B 0,C 180,E1 24421.428,E2 24421.428} C_VEL
LIN {X 0,Y 529.155,Z 598.283,A -85,B 0,C 180,E1 24420.501,E2 24420.501} C_VEL
LIN {X 0,Y 528.017,Z 618.804,A -85,B 0,C 180,E1 24419.37,E2 24419.37} C_VEL
LIN {X 0,Y 526.773,Z 638.707,A -85,B 0,C 180,E1 24418.042,E2 24418.042} C_VEL
LIN {X 0,Y 525.528,Z 658.142,A -85,B 0,C 180,E1 24416.497,E2 24416.497} C_VEL
LIN {X 0,Y 524.353,Z 676.275,A -85,B 0,C 180,E1 24414.803,E2 24414.803} C_VEL
LIN {X 0,Y 523.204,Z 694.223,A -85,B 0,C 180,E1 24412.826,E2 24412.826} C_VEL
LIN {X 0,Y 522.229,Z 710.291,A -85,B 0,C 180,E1 24410.744,E2 24410.744} C_VEL
LIN {X 0,Y 521.444,Z 724.608,A -85,B 0,C 180,E1 24408.56,E2 24408.56} C_VEL
LIN {X 0,Y 520.836,Z 737.279,A -85,B 0,C 180,E1 24406.277,E2 24406.277} C_VEL
LIN {X 0,Y 520.42,Z 748.323,A -85,B 0,C 180,E1 24403.896,E2 24403.896} C_VEL
LIN {X 0,Y 520.159,Z 757.312,A -85,B 0,C 180,E1 24401.532,E2 24401.532} C_VEL
LIN {X 0,Y 520.02,Z 764.402,A -85,B 0,C 180,E1 24399.183,E2 24399.183} C_VEL
LIN {X 0,Y 519.943,Z 770.013,A -85,B 0,C 180,E1 24396.736,E2 24396.736} C_VEL
LIN {X 0,Y 519.917,Z 773.739,A -85,B 0,C 180,E1 24394.412,E2 24394.412} C_VEL
LIN {X 0,Y 519.91,Z 775.904,A -85,B 0,C 180,E1 24391.984,E2 24391.984} C_VEL
LIN {X 0,Y 519.898,Z 776.447,A -85,B 0,C 180,E1 24389.559,E2 24389.559} C_VEL
LIN {X 0,Y 519.913,Z 775.33,A -85,B 0,C 180,E1 24387.134,E2 24387.134} C_VEL
LIN {X 0,Y 519.925,Z 772.492,A -85,B 0,C 180,E1 24384.703,E2 24384.703} C_VEL
LIN {X 0,Y 519.962,Z 767.942,A -85,B 0,C 180,E1 24382.264,E2 24382.264} C_VEL
LIN {X 0,Y 520.064,Z 761.706,A -85,B 0,C 180,E1 24379.85,E2 24379.85} C_VEL
LIN {X 0,Y 520.253,Z 753.861,A -85,B 0,C 180,E1 24377.503,E2 24377.503} C_VEL
LIN {X 0,Y 520.564,Z 744.358,A -85,B 0,C 180,E1 24375.199,E2 24375.199} C_VEL
LIN {X 0,Y 521.037,Z 733.12,A -85,B 0,C 180,E1 24372.926,E2 24372.926} C_VEL
LIN {X 0,Y 521.713,Z 719.628,A -85,B 0,C 180,E1 24370.637,E2 24370.637} C_VEL
LIN {X 0,Y 522.581,Z 704.348,A -85,B 0,C 180,E1 24368.447,E2 24368.447} C_VEL
LIN {X 0,Y 523.601,Z 687.826,A -85,B 0,C 180,E1 24366.433,E2 24366.433} C_VEL
LIN {X 0,Y 524.757,Z 669.937,A -85,B 0,C 180,E1 24364.574,E2 24364.574} C_VEL
LIN {X 0,Y 525.969,Z 651.141,A -85,B 0,C 180,E1 24362.916,E2 24362.916} C_VEL
LIN {X 0,Y 527.241,Z 631.51,A -85,B 0,C 180,E1 24361.452,E2 24361.452} C_VEL
LIN {X 0,Y 528.4,Z 611.755,A -85,B 0,C 180,E1 24360.217,E2 24360.217} C_VEL
LIN {X 0,Y 529.542,Z 591.156,A -85,B 0,C 180,E1 24359.16,E2 24359.16} C_VEL
LIN {X 0,Y 530.522,Z 569.583,A -85,B 0,C 180,E1 24358.28,E2 24358.28} C_VEL
LIN {X 0,Y 531.35,Z 547.824,A -85,B 0,C 180,E1 24357.612,E2 24357.612} C_VEL
LIN {X 0,Y 531.91,Z 525.523,A -85,B 0,C 180,E1 24357.138,E2 24357.138} C_VEL
LIN {X 0,Y 532.749,Z 463.166,A -85,B 0,C 180,E1 24356.172,E2 24356.172} C_VEL
LIN {X 0,Y 535.691,Z 450.286,A -85,B 0,C 180,E1 24355.713,E2 24355.713} C_VEL
LIN {X 0,Y 539.742,Z 433.74,A -85,B 0,C 180,E1 24355.369,E2 24355.369} C_VEL
LIN {X 0,Y 542.931,Z 420.053,A -85,B 0,C 180,E1 24354.905,E2 24354.905} C_VEL
LIN {X 0,Y 547.43,Z 400.742,A -85,B 0,C 180,E1 24354.528,E2 24354.528} C_VEL
LIN {X 0,Y 552.438,Z 375.277,A -85,B 0,C 180,E1 24354.249,E2 24354.249} C_VEL
LIN {X 0,Y 556.055,Z 348.381,A -85,B 0,C 180,E1 24354.001,E2 24354.001} C_VEL
LIN {X 0,Y 558.217,Z 339.22,A -85,B 0,C 180,E1 24353.698,E2 24353.698} C_VEL
LIN {X 0,Y 561.388,Z 318.051,A -85,B 0,C 180,E1 24353.282,E2 24353.282} C_VEL
LIN {X 0,Y 565.601,Z 278.387,A -85,B 0,C 180,E1 24352.714,E2 24352.714} C_VEL
LIN {X 0,Y 568.452,Z 246.769,A -85,B 0,C 180,E1 24352.338,E2 24352.338} C_VEL
LIN {X 0,Y 572.292,Z 236.468,A -85,B 0,C 180,E1 24351.842,E2 24351.842} C_VEL
LIN {X 0,Y 579.388,Z 243.245,A -85,B 0,C 180,E1 24350.958,E2 24350.958} C_VEL
LIN {X 0,Y 583.039,Z 246.192,A -85,B 0,C 180,E1 24350.425,E2 24350.425} C_VEL
LIN {X 0,Y 585.026,Z 248.318,A -85,B 0,C 180,E1 24349.842,E2 24349.842} C_VEL
LIN {X 0,Y 585.543,Z 249.594,A -85,B 0,C 180,E1 24349.285,E2 24349.285} C_VEL
LIN {X 0,Y 584.732,Z 250.244,A -85,B 0,C 180,E1 24348.648,E2 24348.648} C_VEL
LIN {X 0,Y 582.257,Z 250.651,A -85,B 0,C 180,E1 24348.035,E2 24348.035} C_VEL
LIN {X 0,Y 578.529,Z 250.032,A -85,B 0,C 180,E1 24347.487,E2 24347.487} C_VEL
LIN {X 0,Y 573.174,Z 248.046,A -85,B 0,C 180,E1 24346.963,E2 24346.963} C_VEL
LIN {X 0,Y 564.646,Z 243.256,A -85,B 0,C 180,E1 24346.112,E2 24346.112} C_VEL
LIN {X 0,Y 552.062,Z 233.374,A -85,B 0,C 180,E1 24344.645,E2 24344.645} C_VEL
LIN {X 0,Y 545.536,Z 225.708,A -85,B 0,C 180,E1 24343.706,E2 24343.706} C_VEL
LIN {X 0,Y 538.983,Z 213.671,A -85,B 0,C 180,E1 24342.473,E2 24342.473} C_VEL
LIN {X 0,Y 529.764,Z 194.628,A -85,B 0,C 180,E1 24340.482,E2 24340.482} C_VEL
LIN {X 0,Y 522.523,Z 181.215,A -85,B 0,C 180,E1 24338.875,E2 24338.875} C_VEL
LIN {X 0,Y 520.752,Z 177.946,A -85,B 0,C 180,E1 24338.468,E2 24338.468} C_VEL
LIN {X 0,Y 520.547,Z 176.884,A -85,B 0,C 180,E1 24338.346,E2 24338.346} C_VEL
LIN {X 0,Y 520.558,Z 176.887,A -85,B 0,C 180,E1 24334.899,E2 24334.899} C_VEL
LIN {X 0,Y 520.56,Z 176.976,A -85,B 0,C 180,E1 24332.812,E2 24332.812} C_VEL
LIN {X 0,Y 523.219,Z 186.727,A -85,B 0,C 180,E1 24332.025,E2 24332.025} C_VEL
LIN {X 0,Y 524.177,Z 221.525,A -85,B 0,C 180,E1 24329.48,E2 24329.48} C_VEL
LIN {X 0,Y 524.625,Z 252.022,A -85,B 0,C 180,E1 24327.097,E2 24327.097} C_VEL
LIN {X 0,Y 524.65,Z 289.492,A -85,B 0,C 180,E1 24324.009,E2 24324.009} C_VEL
LIN {X 0,Y 524.301,Z 322.622,A -85,B 0,C 180,E1 24321.192,E2 24321.192} C_VEL
LIN {X 0,Y 523.492,Z 456.419,A -85,B 0,C 180,E1 24319.256,E2 24319.256} C_VEL
LIN {X 0,Y 523.39,Z 491.065,A -85,B 0,C 180,E1 24318.741,E2 24318.741} C_VEL
LIN {X 0,Y 523.27,Z 508.499,A -85,B 0,C 180,E1 24318.266,E2 24318.266} C_VEL
LIN {X 0,Y 523.007,Z 525.648,A -85,B 0,C 180,E1 24317.581,E2 24317.581} C_VEL
LIN {X 0,Y 522.673,Z 541.443,A -85,B 0,C 180,E1 24316.732,E2 24316.732} C_VEL
LIN {X 0,Y 522.268,Z 556.068,A -85,B 0,C 180,E1 24315.717,E2 24315.717} C_VEL
LIN {X 0,Y 521.813,Z 570.292,A -85,B 0,C 180,E1 24314.48,E2 24314.48} C_VEL
LIN {X 0,Y 521.407,Z 582.308,A -85,B 0,C 180,E1 24313.191,E2 24313.191} C_VEL
LIN {X 0,Y 521.01,Z 593.334,A -85,B 0,C 180,E1 24311.737,E2 24311.737} C_VEL
LIN {X 0,Y 520.679,Z 602.881,A -85,B 0,C 180,E1 24310.175,E2 24310.175} C_VEL
LIN {X 0,Y 520.426,Z 611.525,A -85,B 0,C 180,E1 24308.396,E2 24308.396} C_VEL
LIN {X 0,Y 520.253,Z 618.158,A -85,B 0,C 180,E1 24306.621,E2 24306.621} C_VEL
LIN {X 0,Y 520.133,Z 623.21,A -85,B 0,C 180,E1 24304.741,E2 24304.741} C_VEL
LIN {X 0,Y 520.071,Z 626.657,A -85,B 0,C 180,E1 24302.755,E2 24302.755} C_VEL
LIN {X 0,Y 520.049,Z 628.277,A -85,B 0,C 180,E1 24300.771,E2 24300.771} C_VEL
LIN {X 0,Y 520.044,Z 628.047,A -85,B 0,C 180,E1 24298.788,E2 24298.788} C_VEL
LIN {X 0,Y 520.061,Z 626.041,A -85,B 0,C 180,E1 24296.803,E2 24296.803} C_VEL
LIN {X 0,Y 520.108,Z 622.444,A -85,B 0,C 180,E1 24294.926,E2 24294.926} C_VEL
LIN {X 0,Y 520.211,Z 616.984,A -85,B 0,C 180,E1 24293.045,E2 24293.045} C_VEL
LIN {X 0,Y 520.396,Z 609.516,A -85,B 0,C 180,E1 24291.158,E2 24291.158} C_VEL
LIN {X 0,Y 520.642,Z 600.991,A -85,B 0,C 180,E1 24289.488,E2 24289.488} C_VEL
LIN {X 0,Y 520.966,Z 590.966,A -85,B 0,C 180,E1 24287.924,E2 24287.924} C_VEL
LIN {X 0,Y 521.39,Z 578.981,A -85,B 0,C 180,E1 24286.413,E2 24286.413} C_VEL
LIN {X 0,Y 521.851,Z 565.817,A -85,B 0,C 180,E1 24285.066,E2 24285.066} C_VEL
LIN {X 0,Y 522.311,Z 551.461,A -85,B 0,C 180,E1 24283.884,E2 24283.884} C_VEL
LIN {X 0,Y 522.767,Z 535.941,A -85,B 0,C 180,E1 24282.869,E2 24282.869} C_VEL
LIN {X 0,Y 523.125,Z 520.412,A -85,B 0,C 180,E1 24282.078,E2 24282.078} C_VEL
LIN {X 0,Y 523.452,Z 503.511,A -85,B 0,C 180,E1 24281.437,E2 24281.437} C_VEL
LIN {X 0,Y 523.632,Z 485.982,A -85,B 0,C 180,E1 24280.996,E2 24280.996} C_VEL
LIN {X 0,Y 524.564,Z 322.484,A -85,B 0,C 180,E1 24278.611,E2 24278.611} C_VEL
LIN {X 0,Y 524.194,Z 320.205,A -85,B 0,C 180,E1 24278.562,E2 24278.562} C_VEL
LIN {X 0,Y 523.699,Z 316.832,A -85,B 0,C 180,E1 24278.387,E2 24278.387} C_VEL
LIN {X 0,Y 522.54,Z 313.417,A -85,B 0,C 180,E1 24278.032,E2 24278.032} C_VEL
LIN {X 0,Y 519.339,Z 308.454,A -85,B 0,C 180,E1 24277.397,E2 24277.397} C_VEL
LIN {X 0,Y 517.333,Z 301.322,A -85,B 0,C 180,E1 24276.62,E2 24276.62} C_VEL
LIN {X 0,Y 516.771,Z 294.52,A -85,B 0,C 180,E1 24275.979,E2 24275.979} C_VEL
LIN {X 0,Y 517.486,Z 258.684,A -85,B 0,C 180,E1 24272.689,E2 24272.689} C_VEL
LIN {X 0,Y 517.993,Z 223.777,A -85,B 0,C 180,E1 24269.492,E2 24269.492} C_VEL
LIN {X 0,Y 518.202,Z 196.172,A -85,B 0,C 180,E1 24266.97,E2 24266.97} C_VEL
LIN {X 0,Y 514.65,Z 184.521,A -85,B 0,C 180,E1 24265.674,E2 24265.674} C_VEL
LIN {X 0,Y 516.698,Z 186.416,A -85,B 0,C 180,E1 24265.459,E2 24265.459} C_VEL
LIN {X 0,Y 518.041,Z 187.312,A -85,B 0,C 180,E1 24265.327,E2 24265.327} C_VEL
LIN {X 0,Y 528.43,Z 204.291,A -85,B 0,C 180,E1 24264.163,E2 24264.163} C_VEL
LIN {X 0,Y 525.617,Z 423.505,A -85,B 0,C 180,E1 24260.787,E2 24260.787} C_VEL
LIN {X 0,Y 525.005,Z 464.715,A -85,B 0,C 180,E1 24260.121,E2 24260.121} C_VEL
LIN {X 0,Y 524.236,Z 485.985,A -85,B 0,C 180,E1 24259.585,E2 24259.585} C_VEL
LIN {X 0,Y 523.29,Z 507.466,A -85,B 0,C 180,E1 24258.836,E2 24258.836} C_VEL
LIN {X 0,Y 522.198,Z 528.045,A -85,B 0,C 180,E1 24257.921,E2 24257.921} C_VEL
LIN {X 0,Y 520.918,Z 548.361,A -85,B 0,C 180,E1 24256.785,E2 24256.785} C_VEL
LIN {X 0,Y 519.683,Z 567.002,A -85,B 0,C 180,E1 24255.545,E2 24255.545} C_VEL
LIN {X 0,Y 518.277,Z 586.703,A -85,B 0,C 180,E1 24253.979,E2 24253.979} C_VEL
LIN {X 0,Y 517.119,Z 602.41,A -85,B 0,C 180,E1 24252.521,E2 24252.521} C_VEL
LIN {X 0,Y 515.891,Z 620.024,A -85,B 0,C 180,E1 24250.633,E2 24250.633} C_VEL
LIN {X 0,Y 514.815,Z 635.583,A -85,B 0,C 180,E1 24248.67,E2 24248.67} C_VEL
LIN {X 0,Y 513.903,Z 650.18,A -85,B 0,C 180,E1 24246.53,E2 24246.53} C_VEL
LIN {X 0,Y 513.222,Z 661.962,A -85,B 0,C 180,E1 24244.503,E2 24244.503} C_VEL
LIN {X 0,Y 512.705,Z 672.973,A -85,B 0,C 180,E1 24242.3,E2 24242.3} C_VEL
LIN {X 0,Y 512.33,Z 682.733,A -85,B 0,C 180,E1 24239.944,E2 24239.944} C_VEL
LIN {X 0,Y 512.114,Z 689.998,A -85,B 0,C 180,E1 24237.816,E2 24237.816} C_VEL
LIN {X 0,Y 511.989,Z 696.86,A -85,B 0,C 180,E1 24235.285,E2 24235.285} C_VEL
LIN {X 0,Y 511.929,Z 701.428,A -85,B 0,C 180,E1 24232.994,E2 24232.994} C_VEL
LIN {X 0,Y 511.904,Z 704.569,A -85,B 0,C 180,E1 24230.675,E2 24230.675} C_VEL
LIN {X 0,Y 511.906,Z 706.234,A -85,B 0,C 180,E1 24228.211,E2 24228.211} C_VEL
LIN {X 0,Y 511.916,Z 706.302,A -85,B 0,C 180,E1 24225.986,E2 24225.986} C_VEL
LIN {X 0,Y 511.915,Z 704.889,A -85,B 0,C 180,E1 24223.555,E2 24223.555} C_VEL
LIN {X 0,Y 511.932,Z 701.817,A -85,B 0,C 180,E1 24221.149,E2 24221.149} C_VEL
LIN {X 0,Y 511.978,Z 697.425,A -85,B 0,C 180,E1 24218.875,E2 24218.875} C_VEL
LIN {X 0,Y 512.105,Z 690.567,A -85,B 0,C 180,E1 24216.277,E2 24216.277} C_VEL
LIN {X 0,Y 512.309,Z 683.378,A -85,B 0,C 180,E1 24214.141,E2 24214.141} C_VEL
LIN {X 0,Y 512.672,Z 673.776,A -85,B 0,C 180,E1 24211.788,E2 24211.788} C_VEL
LIN {X 0,Y 513.183,Z 662.753,A -85,B 0,C 180,E1 24209.554,E2 24209.554} C_VEL
LIN {X 0,Y 513.835,Z 651.194,A -85,B 0,C 180,E1 24207.547,E2 24207.547} C_VEL
LIN {X 0,Y 514.776,Z 636.182,A -85,B 0,C 180,E1 24205.321,E2 24205.321} C_VEL
LIN {X 0,Y 515.789,Z 621.332,A -85,B 0,C 180,E1 24203.433,E2 24203.433} C_VEL
LIN {X 0,Y 517.048,Z 603.469,A -85,B 0,C 180,E1 24201.493,E2 24201.493} C_VEL
LIN {X 0,Y 518.217,Z 587.487,A -85,B 0,C 180,E1 24200,E2 24200} C_VEL
LIN {X 0,Y 519.596,Z 568.285,A -85,B 0,C 180,E1 24198.456,E2 24198.456} C_VEL
LIN {X 0,Y 520.855,Z 549.497,A -85,B 0,C 180,E1 24197.196,E2 24197.196} C_VEL
LIN {X 0,Y 522.052,Z 530.327,A -85,B 0,C 180,E1 24196.107,E2 24196.107} C_VEL
LIN {X 0,Y 523.175,Z 509.631,A -85,B 0,C 180,E1 24195.162,E2 24195.162} C_VEL
LIN {X 0,Y 524.109,Z 489.723,A -85,B 0,C 180,E1 24194.439,E2 24194.439} C_VEL
LIN {X 0,Y 524.865,Z 468.19,A -85,B 0,C 180,E1 24193.866,E2 24193.866} C_VEL
LIN {X 0,Y 525.439,Z 439.176,A -85,B 0,C 180,E1 24193.362,E2 24193.362} C_VEL
LIN {X 0,Y 528.045,Z 231.195,A -85,B 0,C 180,E1 24190.158,E2 24190.158} C_VEL
LIN {X 0,Y 528.286,Z 203.686,A -85,B 0,C 180,E1 24189.714,E2 24189.714} C_VEL
LIN {X 0,Y 517.534,Z 186.624,A -85,B 0,C 180,E1 24188.474,E2 24188.474} C_VEL
LIN {X 0,Y 514.903,Z 182.55,A -85,B 0,C 180,E1 24188.157,E2 24188.157} C_VEL
LIN {X 0,Y 512.978,Z 179.43,A -85,B 0,C 180,E1 24187.921,E2 24187.921} C_VEL
LIN {X 0,Y 512.629,Z 177.881,A -85,B 0,C 180,E1 24187.855,E2 24187.855} C_VEL
LIN {X 0,Y 512.637,Z 177.879,A -85,B 0,C 180,E1 24184.342,E2 24184.342} C_VEL
LIN {X 0,Y 512.648,Z 177.87,A -85,B 0,C 180,E1 24180.817,E2 24180.817} C_VEL
LIN {X 0,Y 512.602,Z 177.879,A -85,B 0,C 180,E1 24177.421,E2 24177.421} C_VEL
LIN {X 0,Y 512.58,Z 177.884,A -85,B 0,C 180,E1 24173.859,E2 24173.859} C_VEL
LIN {X 0,Y 512.616,Z 177.88,A -85,B 0,C 180,E1 24170.395,E2 24170.395} C_VEL
LIN {X 0,Y 512.647,Z 177.878,A -85,B 0,C 180,E1 24167.004,E2 24167.004} C_VEL
LIN {X 0,Y 512.639,Z 177.878,A -85,B 0,C 180,E1 24163.485,E2 24163.485} C_VEL
LIN {X 0,Y 512.637,Z 177.873,A -85,B 0,C 180,E1 24159.958,E2 24159.958} C_VEL
LIN {X 0,Y 512.645,Z 177.87,A -85,B 0,C 180,E1 24156.504,E2 24156.504} C_VEL
LIN {X 0,Y 512.62,Z 177.878,A -85,B 0,C 180,E1 24152.97,E2 24152.97} C_VEL
LIN {X 0,Y 512.609,Z 177.882,A -85,B 0,C 180,E1 24149.57,E2 24149.57} C_VEL
LIN {X 0,Y 512.624,Z 177.876,A -85,B 0,C 180,E1 24146.031,E2 24146.031} C_VEL
LIN {X 0,Y 512.65,Z 177.863,A -85,B 0,C 180,E1 24142.596,E2 24142.596} C_VEL
LIN {X 0,Y 512.619,Z 177.875,A -85,B 0,C 180,E1 24139.129,E2 24139.129} C_VEL
LIN {X 0,Y 512.594,Z 177.882,A -85,B 0,C 180,E1 24135.616,E2 24135.616} C_VEL
LIN {X 0,Y 512.61,Z 177.881,A -85,B 0,C 180,E1 24132.255,E2 24132.255} C_VEL
LIN {X 0,Y 512.646,Z 177.869,A -85,B 0,C 180,E1 24128.864,E2 24128.864} C_VEL
LIN {X 0,Y 512.64,Z 177.876,A -85,B 0,C 180,E1 24125.372,E2 24125.372} C_VEL
LIN {X 0,Y 512.644,Z 177.881,A -85,B 0,C 180,E1 24121.789,E2 24121.789} C_VEL
LIN {X 0,Y 512.65,Z 177.875,A -85,B 0,C 180,E1 24118.324,E2 24118.324} C_VEL
LIN {X 0,Y 512.603,Z 177.876,A -85,B 0,C 180,E1 24114.965,E2 24114.965} C_VEL
LIN {X 0,Y 512.579,Z 177.877,A -85,B 0,C 180,E1 24111.484,E2 24111.484} C_VEL
LIN {X 0,Y 512.618,Z 177.873,A -85,B 0,C 180,E1 24108.068,E2 24108.068} C_VEL
LIN {X 0,Y 512.646,Z 177.872,A -85,B 0,C 180,E1 24104.734,E2 24104.734} C_VEL
LIN {X 0,Y 512.638,Z 177.875,A -85,B 0,C 180,E1 24101.227,E2 24101.227} C_VEL
LIN {X 0,Y 512.646,Z 177.876,A -85,B 0,C 180,E1 24097.767,E2 24097.767} C_VEL
LIN {X 0,Y 512.645,Z 177.878,A -85,B 0,C 180,E1 24094.219,E2 24094.219} C_VEL
LIN {X 0,Y 512.606,Z 177.877,A -85,B 0,C 180,E1 24090.815,E2 24090.815} C_VEL
LIN {X 0,Y 512.643,Z 178.077,A -85,B 0,C 180,E1 24090.047,E2 24090.047} C_VEL
LIN {X 0,Y 513.834,Z 181.272,A -85,B 0,C 180,E1 24089.607,E2 24089.607} C_VEL
LIN {X 0,Y 514.946,Z 183.253,A -85,B 0,C 180,E1 24089.292,E2 24089.292} C_VEL
LIN {X 0,Y 522.785,Z 199.2,A -85,B 0,C 180,E1 24086.97,E2 24086.97} C_VEL
LIN {X 0,Y 529.998,Z 214.7,A -85,B 0,C 180,E1 24084.873,E2 24084.873} C_VEL
LIN {X 0,Y 527.912,Z 256.602,A -85,B 0,C 180,E1 24081.595,E2 24081.595} C_VEL
LIN {X 0,Y 526.974,Z 285.725,A -85,B 0,C 180,E1 24079.327,E2 24079.327} C_VEL
LIN {X 0,Y 528.241,Z 300.298,A -85,B 0,C 180,E1 24078.062,E2 24078.062} C_VEL
LIN {X 0,Y 531.2,Z 312.922,A -85,B 0,C 180,E1 24076.827,E2 24076.827} C_VEL
LIN {X 0,Y 535.424,Z 323.177,A -85,B 0,C 180,E1 24075.701,E2 24075.701} C_VEL
LIN {X 0,Y 540.94,Z 331.762,A -85,B 0,C 180,E1 24074.633,E2 24074.633} C_VEL
LIN {X 0,Y 547.953,Z 339.15,A -85,B 0,C 180,E1 24073.58,E2 24073.58} C_VEL
LIN {X 0,Y 556.508,Z 345.233,A -85,B 0,C 180,E1 24072.555,E2 24072.555} C_VEL
LIN {X 0,Y 565.867,Z 349.593,A -85,B 0,C 180,E1 24071.633,E2 24071.633} C_VEL
LIN {X 0,Y 570.421,Z 350.602,A -85,B 0,C 180,E1 24071.087,E2 24071.087} C_VEL
LIN {X 0,Y 573.544,Z 350.304,A -85,B 0,C 180,E1 24070.529,E2 24070.529} C_VEL
LIN {X 0,Y 575.416,Z 349.076,A -85,B 0,C 180,E1 24069.978,E2 24069.978} C_VEL
LIN {X 0,Y 576.156,Z 346.593,A -85,B 0,C 180,E1 24069.335,E2 24069.335} C_VEL
LIN {X 0,Y 575.338,Z 343.322,A -85,B 0,C 180,E1 24068.76,E2 24068.76} C_VEL
LIN {X 0,Y 573.027,Z 339.294,A -85,B 0,C 180,E1 24068.258,E2 24068.258} C_VEL
LIN {X 0,Y 566.47,Z 329.452,A -85,B 0,C 180,E1 24067.402,E2 24067.402} C_VEL
LIN {X 0,Y 565.126,Z 327.31,A -85,B 0,C 180,E1 24067.223,E2 24067.223} C_VEL
LIN {X 0,Y 562.284,Z 344.544,A -85,B 0,C 180,E1 24066.84,E2 24066.84} C_VEL
LIN {X 0,Y 560.491,Z 352.337,A -85,B 0,C 180,E1 24066.595,E2 24066.595} C_VEL
LIN {X 0,Y 557.215,Z 388.608,A -85,B 0,C 180,E1 24066.194,E2 24066.194} C_VEL
LIN {X 0,Y 553.575,Z 407.648,A -85,B 0,C 180,E1 24066.037,E2 24066.037} C_VEL
LIN {X 0,Y 548.137,Z 426.206,A -85,B 0,C 180,E1 24065.873,E2 24065.873} C_VEL
LIN {X 0,Y 543.349,Z 439.493,A -85,B 0,C 180,E1 24065.621,E2 24065.621} C_VEL
LIN {X 0,Y 540.007,Z 448.771,A -85,B 0,C 180,E1 24065.288,E2 24065.288} C_VEL
LIN {X 0,Y 537.415,Z 455.199,A -85,B 0,C 180,E1 24065.157,E2 24065.157} C_VEL
LIN {X 0,Y 532.797,Z 466.49,A -85,B 0,C 180,E1 24064.85,E2 24064.85} C_VEL
LIN {X 0,Y 528.763,Z 477.639,A -85,B 0,C 180,E1 24064.364,E2 24064.364} C_VEL
LIN {X 0,Y 525.735,Z 486.389,A -85,B 0,C 180,E1 24063.947,E2 24063.947} C_VEL
LIN {X 0,Y 525.003,Z 534.267,A -85,B 0,C 180,E1 24063.174,E2 24063.174} C_VEL
LIN {X 0,Y 524.226,Z 556.368,A -85,B 0,C 180,E1 24062.619,E2 24062.619} C_VEL
LIN {X 0,Y 523.285,Z 578.071,A -85,B 0,C 180,E1 24061.86,E2 24061.86} C_VEL
LIN {X 0,Y 522.148,Z 598.904,A -85,B 0,C 180,E1 24060.922,E2 24060.922} C_VEL
LIN {X 0,Y 520.864,Z 619.771,A -85,B 0,C 180,E1 24059.75,E2 24059.75} C_VEL
LIN {X 0,Y 519.48,Z 639.784,A -85,B 0,C 180,E1 24058.386,E2 24058.386} C_VEL
LIN {X 0,Y 518.067,Z 659.791,A -85,B 0,C 180,E1 24056.758,E2 24056.758} C_VEL
LIN {X 0,Y 516.795,Z 677.395,A -85,B 0,C 180,E1 24055.069,E2 24055.069} C_VEL
LIN {X 0,Y 515.565,Z 694.696,A -85,B 0,C 180,E1 24053.124,E2 24053.124} C_VEL
LIN {X 0,Y 514.513,Z 710.292,A -85,B 0,C 180,E1 24051.07,E2 24051.07} C_VEL
LIN {X 0,Y 513.642,Z 724.612,A -85,B 0,C 180,E1 24048.853,E2 24048.853} C_VEL
LIN {X 0,Y 512.963,Z 737.283,A -85,B 0,C 180,E1 24046.534,E2 24046.534} C_VEL
LIN {X 0,Y 512.488,Z 748.326,A -85,B 0,C 180,E1 24044.115,E2 24044.115} C_VEL
LIN {X 0,Y 512.19,Z 757.312,A -85,B 0,C 180,E1 24041.714,E2 24041.714} C_VEL
LIN {X 0,Y 512.031,Z 764.403,A -85,B 0,C 180,E1 24039.327,E2 24039.327} C_VEL
LIN {X 0,Y 511.95,Z 770.014,A -85,B 0,C 180,E1 24036.842,E2 24036.842} C_VEL
LIN {X 0,Y 511.919,Z 773.74,A -85,B 0,C 180,E1 24034.481,E2 24034.481} C_VEL
LIN {X 0,Y 511.911,Z 775.906,A -85,B 0,C 180,E1 24032.015,E2 24032.015} C_VEL
LIN {X 0,Y 511.898,Z 776.447,A -85,B 0,C 180,E1 24029.552,E2 24029.552} C_VEL
LIN {X 0,Y 511.914,Z 775.329,A -85,B 0,C 180,E1 24027.089,E2 24027.089} C_VEL
LIN {X 0,Y 511.926,Z 772.495,A -85,B 0,C 180,E1 24024.62,E2 24024.62} C_VEL
LIN {X 0,Y 511.973,Z 767.945,A -85,B 0,C 180,E1 24022.142,E2 24022.142} C_VEL
LIN {X 0,Y 512.082,Z 761.908,A -85,B 0,C 180,E1 24019.761,E2 24019.761} C_VEL
LIN {X 0,Y 512.29,Z 754.106,A -85,B 0,C 180,E1 24017.373,E2 24017.373} C_VEL
LIN {X 0,Y 512.645,Z 744.361,A -85,B 0,C 180,E1 24014.965,E2 24014.965} C_VEL
LIN {X 0,Y 513.177,Z 733.121,A -85,B 0,C 180,E1 24012.656,E2 24012.656} C_VEL
LIN {X 0,Y 513.944,Z 719.564,A -85,B 0,C 180,E1 24010.322,E2 24010.322} C_VEL
LIN {X 0,Y 514.908,Z 704.351,A -85,B 0,C 180,E1 24008.11,E2 24008.11} C_VEL
LIN {X 0,Y 516.056,Z 687.701,A -85,B 0,C 180,E1 24006.052,E2 24006.052} C_VEL
LIN {X 0,Y 517.373,Z 669.481,A -85,B 0,C 180,E1 24004.138,E2 24004.138} C_VEL
LIN {X 0,Y 518.711,Z 650.602,A -85,B 0,C 180,E1 24002.46,E2 24002.46} C_VEL
LIN {X 0,Y 520.129,Z 630.615,A -85,B 0,C 180,E1 24000.959,E2 24000.959} C_VEL
LIN {X 0,Y 521.427,Z 610.741,A -85,B 0,C 180,E1 23999.714,E2 23999.714} C_VEL
LIN {X 0,Y 522.667,Z 589.894,A -85,B 0,C 180,E1 23998.645,E2 23998.645} C_VEL
LIN {X 0,Y 523.752,Z 568.055,A -85,B 0,C 180,E1 23997.764,E2 23997.764} C_VEL
LIN {X 0,Y 524.619,Z 546.35,A -85,B 0,C 180,E1 23997.104,E2 23997.104} C_VEL
LIN {X 0,Y 525.237,Z 523.591,A -85,B 0,C 180,E1 23996.63,E2 23996.63} C_VEL
LIN {X 0,Y 525.817,Z 481.624,A -85,B 0,C 180,E1 23995.977,E2 23995.977} C_VEL
LIN {X 0,Y 528.961,Z 468.02,A -85,B 0,C 180,E1 23995.486,E2 23995.486} C_VEL
LIN {X 0,Y 533.232,Z 450.364,A -85,B 0,C 180,E1 23994.887,E2 23994.887} C_VEL
LIN {X 0,Y 538.056,Z 433.51,A -85,B 0,C 180,E1 23994.499,E2 23994.499} C_VEL
LIN {X 0,Y 541.159,Z 420.835,A -85,B 0,C 180,E1 23994.082,E2 23994.082} C_VEL
LIN {X 0,Y 546.668,Z 401.255,A -85,B 0,C 180,E1 23993.695,E2 23993.695} C_VEL
LIN {X 0,Y 553.391,Z 376.134,A -85,B 0,C 180,E1 23993.431,E2 23993.431} C_VEL
LIN {X 0,Y 558.784,Z 350.684,A -85,B 0,C 180,E1 23993.25,E2 23993.25} C_VEL
LIN {X 0,Y 561.319,Z 339.925,A -85,B 0,C 180,E1 23992.929,E2 23992.929} C_VEL
LIN {X 0,Y 565.644,Z 317.269,A -85,B 0,C 180,E1 23992.555,E2 23992.555} C_VEL
LIN {X 0,Y 569.692,Z 287.162,A -85,B 0,C 180,E1 23992.176,E2 23992.176} C_VEL
LIN {X 0,Y 573.142,Z 249.791,A -85,B 0,C 180,E1 23991.734,E2 23991.734} C_VEL
LIN {X 0,Y 574.072,Z 247.762,A -85,B 0,C 180,E1 23991.617,E2 23991.617} C_VEL
LIN {X 0,Y 580.292,Z 252.875,A -85,B 0,C 180,E1 23990.808,E2 23990.808} C_VEL
LIN {X 0,Y 582.677,Z 255.196,A -85,B 0,C 180,E1 23990.242,E2 23990.242} C_VEL
LIN {X 0,Y 583.564,Z 256.823,A -85,B 0,C 180,E1 23989.635,E2 23989.635} C_VEL
LIN {X 0,Y 582.982,Z 257.716,A -85,B 0,C 180,E1 23988.993,E2 23988.993} C_VEL
LIN {X 0,Y 581.191,Z 258.064,A -85,B 0,C 180,E1 23988.448,E2 23988.448} C_VEL
LIN {X 0,Y 578.015,Z 257.929,A -85,B 0,C 180,E1 23987.909,E2 23987.909} C_VEL
LIN {X 0,Y 574.03,Z 256.882,A -85,B 0,C 180,E1 23987.458,E2 23987.458} C_VEL
LIN {X 0,Y 564.49,Z 252.581,A -85,B 0,C 180,E1 23986.57,E2 23986.57} C_VEL
LIN {X 0,Y 552.892,Z 244.488,A -85,B 0,C 180,E1 23985.292,E2 23985.292} C_VEL
LIN {X 0,Y 545.206,Z 237.67,A -85,B 0,C 180,E1 23984.324,E2 23984.324} C_VEL
LIN {X 0,Y 538.888,Z 229.555,A -85,B 0,C 180,E1 23983.354,E2 23983.354} C_VEL
LIN {X 0,Y 523.902,Z 199.431,A -85,B 0,C 180,E1 23980.17,E2 23980.17} C_VEL
LIN {X 0,Y 517.184,Z 186.851,A -85,B 0,C 180,E1 23978.641,E2 23978.641} C_VEL
LIN {X 0,Y 514.521,Z 182.128,A -85,B 0,C 180,E1 23978.026,E2 23978.026} C_VEL
LIN {X 0,Y 512.84,Z 178.876,A -85,B 0,C 180,E1 23977.607,E2 23977.607} C_VEL
LIN {X 0,Y 512.649,Z 177.871,A -85,B 0,C 180,E1 23977.482,E2 23977.482} C_VEL
LIN {X 0,Y 512.62,Z 177.881,A -85,B 0,C 180,E1 23974.008,E2 23974.008} C_VEL
LIN {X 0,Y 512.66,Z 178.057,A -85,B 0,C 180,E1 23973.14,E2 23973.14} C_VEL
LIN {X 0,Y 515.772,Z 189.341,A -85,B 0,C 180,E1 23972.215,E2 23972.215} C_VEL
LIN {X 0,Y 516.725,Z 223.805,A -85,B 0,C 180,E1 23969.693,E2 23969.693} C_VEL
LIN {X 0,Y 517.181,Z 254.047,A -85,B 0,C 180,E1 23967.332,E2 23967.332} C_VEL
LIN {X 0,Y 517.225,Z 288.569,A -85,B 0,C 180,E1 23964.497,E2 23964.497} C_VEL
LIN {X 0,Y 516.825,Z 323.828,A -85,B 0,C 180,E1 23961.478,E2 23961.478} C_VEL
LIN {X 0,Y 515.931,Z 433.781,A -85,B 0,C 180,E1 23959.819,E2 23959.819} C_VEL
LIN {X 0,Y 515.679,Z 491.976,A -85,B 0,C 180,E1 23958.962,E2 23958.962} C_VEL
LIN {X 0,Y 515.584,Z 509.238,A -85,B 0,C 180,E1 23958.497,E2 23958.497} C_VEL
LIN {X 0,Y 515.343,Z 525.578,A -85,B 0,C 180,E1 23957.851,E2 23957.851} C_VEL
LIN {X 0,Y 514.999,Z 541.793,A -85,B 0,C 180,E1 23956.989,E2 23956.989} C_VEL
LIN {X 0,Y 514.587,Z 556.768,A -85,B 0,C 180,E1 23955.958,E2 23955.958} C_VEL
LIN {X 0,Y 514.128,Z 570.589,A -85,B 0,C 180,E1 23954.759,E2 23954.759} C_VEL
LIN {X 0,Y 513.674,Z 583.336,A -85,B 0,C 180,E1 23953.393,E2 23953.393} C_VEL
LIN {X 0,Y 513.252,Z 594.503,A -85,B 0,C 180,E1 23951.917,E2 23951.917} C_VEL
LIN {X 0,Y 512.891,Z 604.124,A -85,B 0,C 180,E1 23950.332,E2 23950.332} C_VEL
LIN {X 0,Y 512.607,Z 612.822,A -85,B 0,C 180,E1 23948.525,E2 23948.525} C_VEL
LIN {X 0,Y 512.408,Z 619.639,A -85,B 0,C 180,E1 23946.678,E2 23946.678} C_VEL
LIN {X 0,Y 512.272,Z 624.572,A -85,B 0,C 180,E1 23944.814,E2 23944.814} C_VEL
LIN {X 0,Y 512.195,Z 628.018,A -85,B 0,C 180,E1 23942.797,E2 23942.797} C_VEL
LIN {X 0,Y 512.164,Z 629.628,A -85,B 0,C 180,E1 23940.783,E2 23940.783} C_VEL
LIN {X 0,Y 512.154,Z 629.363,A -85,B 0,C 180,E1 23938.769,E2 23938.769} C_VEL
LIN {X 0,Y 512.176,Z 627.246,A -85,B 0,C 180,E1 23936.701,E2 23936.701} C_VEL
LIN {X 0,Y 512.233,Z 623.386,A -85,B 0,C 180,E1 23934.736,E2 23934.736} C_VEL
LIN {X 0,Y 512.352,Z 617.755,A -85,B 0,C 180,E1 23932.825,E2 23932.825} C_VEL
LIN {X 0,Y 512.548,Z 610.605,A -85,B 0,C 180,E1 23931.021,E2 23931.021} C_VEL
LIN {X 0,Y 512.822,Z 601.933,A -85,B 0,C 180,E1 23929.316,E2 23929.316} C_VEL
LIN {X 0,Y 513.174,Z 591.865,A -85,B 0,C 180,E1 23927.738,E2 23927.738} C_VEL
LIN {X 0,Y 513.631,Z 579.765,A -85,B 0,C 180,E1 23926.204,E2 23926.204} C_VEL
LIN {X 0,Y 514.129,Z 566.478,A -85,B 0,C 180,E1 23924.836,E2 23924.836} C_VEL
LIN {X 0,Y 514.619,Z 551.925,A -85,B 0,C 180,E1 23923.637,E2 23923.637} C_VEL
LIN {X 0,Y 515.103,Z 536.202,A -85,B 0,C 180,E1 23922.606,E2 23922.606} C_VEL
LIN {X 0,Y 515.5,Z 519.781,A -85,B 0,C 180,E1 23921.774,E2 23921.774} C_VEL
LIN {X 0,Y 515.812,Z 502.61,A -85,B 0,C 180,E1 23921.145,E2 23921.145} C_VEL
LIN {X 0,Y 515.994,Z 484.375,A -85,B 0,C 180,E1 23920.705,E2 23920.705} C_VEL
LIN {X 0,Y 517.095,Z 323.738,A -85,B 0,C 180,E1 23918.323,E2 23918.323} C_VEL
LIN {X 0,Y 516.296,Z 318.937,A -85,B 0,C 180,E1 23918.215,E2 23918.215} C_VEL
LIN {X 0,Y 516.771,Z 294.52,A -85,B 0,C 180,E1 23915.979,E2 23915.979} C_VEL
LIN {X 0,Y 515.944,Z 288.823,A -85,B 0,C 180,E1 23915.402,E2 23915.402} C_VEL
LIN {X 0,Y 510.402,Z 274.506,A -85,B 0,C 180,E1 23913.762,E2 23913.762} C_VEL
LIN {X 0,Y 509.818,Z 269.499,A -85,B 0,C 180,E1 23913.264,E2 23913.264} C_VEL
LIN {X 0,Y 510.456,Z 232.98,A -85,B 0,C 180,E1 23909.904,E2 23909.904} C_VEL
LIN {X 0,Y 510.822,Z 198.805,A -85,B 0,C 180,E1 23906.766,E2 23906.766} C_VEL
LIN {X 0,Y 509.004,Z 192.523,A -85,B 0,C 180,E1 23906.04,E2 23906.04} C_VEL
LIN {X 0,Y 510.948,Z 194.319,A -85,B 0,C 180,E1 23905.831,E2 23905.831} C_VEL
LIN {X 0,Y 513.372,Z 194.558,A -85,B 0,C 180,E1 23905.61,E2 23905.61} C_VEL
LIN {X 0,Y 514.083,Z 194.611,A -85,B 0,C 180,E1 23905.546,E2 23905.546} C_VEL
LIN {X 0,Y 521.994,Z 207.356,A -85,B 0,C 180,E1 23904.645,E2 23904.645} C_VEL
LIN {X 0,Y 518.992,Z 422.204,A -85,B 0,C 180,E1 23901.3,E2 23901.3} C_VEL
LIN {X 0,Y 518.31,Z 464.64,A -85,B 0,C 180,E1 23900.608,E2 23900.608} C_VEL
LIN {X 0,Y 517.489,Z 485.844,A -85,B 0,C 180,E1 23900.069,E2 23900.069} C_VEL
LIN {X 0,Y 516.453,Z 507.329,A -85,B 0,C 180,E1 23899.315,E2 23899.315} C_VEL
LIN {X 0,Y 515.263,Z 528.039,A -85,B 0,C 180,E1 23898.385,E2 23898.385} C_VEL
LIN {X 0,Y 513.88,Z 548.031,A -85,B 0,C 180,E1 23897.258,E2 23897.258} C_VEL
LIN {X 0,Y 512.645,Z 565.192,A -85,B 0,C 180,E1 23896.11,E2 23896.11} C_VEL
LIN {X 0,Y 511.156,Z 584.418,A -85,B 0,C 180,E1 23894.601,E2 23894.601} C_VEL
LIN {X 0,Y 509.806,Z 601.195,A -85,B 0,C 180,E1 23893.041,E2 23893.041} C_VEL
LIN {X 0,Y 508.551,Z 617.38,A -85,B 0,C 180,E1 23891.318,E2 23891.318} C_VEL
LIN {X 0,Y 507.304,Z 633.361,A -85,B 0,C 180,E1 23889.317,E2 23889.317} C_VEL
LIN {X 0,Y 506.352,Z 646.843,A -85,B 0,C 180,E1 23887.369,E2 23887.369} C_VEL
LIN {X 0,Y 505.479,Z 660.683,A -85,B 0,C 180,E1 23885.023,E2 23885.023} C_VEL
LIN {X 0,Y 504.891,Z 671.511,A -85,B 0,C 180,E1 23882.862,E2 23882.862} C_VEL
LIN {X 0,Y 504.417,Z 681.965,A -85,B 0,C 180,E1 23880.362,E2 23880.362} C_VEL
LIN {X 0,Y 504.159,Z 689.452,A -85,B 0,C 180,E1 23878.165,E2 23878.165} C_VEL
LIN {X 0,Y 504.004,Z 696.124,A -85,B 0,C 180,E1 23875.751,E2 23875.751} C_VEL
LIN {X 0,Y 503.939,Z 701.149,A -85,B 0,C 180,E1 23873.256,E2 23873.256} C_VEL
LIN {X 0,Y 503.906,Z 704.502,A -85,B 0,C 180,E1 23870.804,E2 23870.804} C_VEL
LIN {X 0,Y 503.904,Z 706.222,A -85,B 0,C 180,E1 23868.271,E2 23868.271} C_VEL
LIN {X 0,Y 503.916,Z 706.309,A -85,B 0,C 180,E1 23866.01,E2 23866.01} C_VEL
LIN {X 0,Y 503.914,Z 704.917,A -85,B 0,C 180,E1 23863.527,E2 23863.527} C_VEL
LIN {X 0,Y 503.933,Z 701.878,A -85,B 0,C 180,E1 23861.097,E2 23861.097} C_VEL
LIN {X 0,Y 503.984,Z 697.514,A -85,B 0,C 180,E1 23858.787,E2 23858.787} C_VEL
LIN {X 0,Y 504.12,Z 691.047,A -85,B 0,C 180,E1 23856.263,E2 23856.263} C_VEL
LIN {X 0,Y 504.354,Z 683.531,A -85,B 0,C 180,E1 23853.979,E2 23853.979} C_VEL
LIN {X 0,Y 504.76,Z 673.977,A -85,B 0,C 180,E1 23851.589,E2 23851.589} C_VEL
LIN {X 0,Y 505.326,Z 662.989,A -85,B 0,C 180,E1 23849.32,E2 23849.32} C_VEL
LIN {X 0,Y 506.046,Z 651.468,A -85,B 0,C 180,E1 23847.282,E2 23847.282} C_VEL
LIN {X 0,Y 507.086,Z 636.514,A -85,B 0,C 180,E1 23845.023,E2 23845.023} C_VEL
LIN {X 0,Y 508.202,Z 621.699,A -85,B 0,C 180,E1 23843.107,E2 23843.107} C_VEL
LIN {X 0,Y 509.59,Z 603.919,A -85,B 0,C 180,E1 23841.14,E2 23841.14} C_VEL
LIN {X 0,Y 510.829,Z 588.399,A -85,B 0,C 180,E1 23839.664,E2 23839.664} C_VEL
LIN {X 0,Y 512.317,Z 569.618,A -85,B 0,C 180,E1 23838.118,E2 23838.118} C_VEL
LIN {X 0,Y 513.689,Z 550.956,A -85,B 0,C 180,E1 23836.837,E2 23836.837} C_VEL
LIN {X 0,Y 514.919,Z 532.839,A -85,B 0,C 180,E1 23835.781,E2 23835.781} C_VEL
LIN {X 0,Y 516.273,Z 510.607,A -85,B 0,C 180,E1 23834.729,E2 23834.729} C_VEL
LIN {X 0,Y 517.292,Z 490.551,A -85,B 0,C 180,E1 23833.987,E2 23833.987} C_VEL
LIN {X 0,Y 518.132,Z 468.935,A -85,B 0,C 180,E1 23833.398,E2 23833.398} C_VEL
LIN {X 0,Y 518.746,Z 441.782,A -85,B 0,C 180,E1 23832.912,E2 23832.912} C_VEL
LIN {X 0,Y 521.547,Z 239.944,A -85,B 0,C 180,E1 23829.762,E2 23829.762} C_VEL
LIN {X 0,Y 522.014,Z 207.062,A -85,B 0,C 180,E1 23829.23,E2 23829.23} C_VEL
LIN {X 0,Y 510.381,Z 188.546,A -85,B 0,C 180,E1 23827.842,E2 23827.842} C_VEL
LIN {X 0,Y 507.714,Z 184.294,A -85,B 0,C 180,E1 23827.508,E2 23827.508} C_VEL
LIN {X 0,Y 505.305,Z 181.057,A -85,B 0,C 180,E1 23827.214,E2 23827.214} C_VEL
LIN {X 0,Y 504.708,Z 178.865,A -85,B 0,C 180,E1 23827.103,E2 23827.103} C_VEL
LIN {X 0,Y 504.696,Z 178.862,A -85,B 0,C 180,E1 23823.529,E2 23823.529} C_VEL
LIN {X 0,Y 504.695,Z 178.868,A -85,B 0,C 180,E1 23820.05,E2 23820.05} C_VEL
LIN {X 0,Y 504.697,Z 178.87,A -85,B 0,C 180,E1 23816.518,E2 23816.518} C_VEL
LIN {X 0,Y 504.694,Z 178.868,A -85,B 0,C 180,E1 23812.968,E2 23812.968} C_VEL
LIN {X 0,Y 504.683,Z 178.872,A -85,B 0,C 180,E1 23809.533,E2 23809.533} C_VEL
LIN {X 0,Y 504.69,Z 178.869,A -85,B 0,C 180,E1 23806.1,E2 23806.1} C_VEL
LIN {X 0,Y 504.706,Z 178.865,A -85,B 0,C 180,E1 23802.527,E2 23802.527} C_VEL
LIN {X 0,Y 504.686,Z 178.866,A -85,B 0,C 180,E1 23799.049,E2 23799.049} C_VEL
LIN {X 0,Y 504.65,Z 178.867,A -85,B 0,C 180,E1 23795.627,E2 23795.627} C_VEL
LIN {X 0,Y 504.653,Z 178.86,A -85,B 0,C 180,E1 23792.072,E2 23792.072} C_VEL
LIN {X 0,Y 504.713,Z 178.861,A -85,B 0,C 180,E1 23788.777,E2 23788.777} C_VEL
LIN {X 0,Y 504.706,Z 178.868,A -85,B 0,C 180,E1 23785.21,E2 23785.21} C_VEL
LIN {X 0,Y 504.706,Z 178.862,A -85,B 0,C 180,E1 23781.702,E2 23781.702} C_VEL
LIN {X 0,Y 504.704,Z 178.857,A -85,B 0,C 180,E1 23778.122,E2 23778.122} C_VEL
LIN {X 0,Y 504.706,Z 178.864,A -85,B 0,C 180,E1 23774.572,E2 23774.572} C_VEL
LIN {X 0,Y 504.683,Z 178.872,A -85,B 0,C 180,E1 23770.964,E2 23770.964} C_VEL
LIN {X 0,Y 504.677,Z 178.864,A -85,B 0,C 180,E1 23767.514,E2 23767.514} C_VEL
LIN {X 0,Y 504.692,Z 178.856,A -85,B 0,C 180,E1 23763.976,E2 23763.976} C_VEL
LIN {X 0,Y 504.711,Z 178.86,A -85,B 0,C 180,E1 23760.454,E2 23760.454} C_VEL
LIN {X 0,Y 504.672,Z 178.868,A -85,B 0,C 180,E1 23757.048,E2 23757.048} C_VEL
LIN {X 0,Y 504.643,Z 178.873,A -85,B 0,C 180,E1 23753.516,E2 23753.516} C_VEL
LIN {X 0,Y 504.672,Z 178.871,A -85,B 0,C 180,E1 23750.075,E2 23750.075} C_VEL
LIN {X 0,Y 504.713,Z 178.867,A -85,B 0,C 180,E1 23746.579,E2 23746.579} C_VEL
LIN {X 0,Y 504.704,Z 178.868,A -85,B 0,C 180,E1 23743.069,E2 23743.069} C_VEL
LIN {X 0,Y 504.704,Z 178.864,A -85,B 0,C 180,E1 23739.562,E2 23739.562} C_VEL
LIN {X 0,Y 504.709,Z 178.86,A -85,B 0,C 180,E1 23736.039,E2 23736.039} C_VEL
LIN {X 0,Y 504.684,Z 178.867,A -85,B 0,C 180,E1 23732.509,E2 23732.509} C_VEL
LIN {X 0,Y 504.676,Z 179.006,A -85,B 0,C 180,E1 23730.944,E2 23730.944} C_VEL
LIN {X 0,Y 505.804,Z 182.036,A -85,B 0,C 180,E1 23730.514,E2 23730.514} C_VEL
LIN {X 0,Y 506.939,Z 183.911,A -85,B 0,C 180,E1 23730.197,E2 23730.197} C_VEL
LIN {X 0,Y 515.345,Z 201.133,A -85,B 0,C 180,E1 23727.623,E2 23727.623} C_VEL
LIN {X 0,Y 523.513,Z 218.722,A -85,B 0,C 180,E1 23725.198,E2 23725.198} C_VEL
LIN {X 0,Y 521.284,Z 260.188,A -85,B 0,C 180,E1 23721.928,E2 23721.928} C_VEL
LIN {X 0,Y 520.287,Z 288.229,A -85,B 0,C 180,E1 23719.723,E2 23719.723} C_VEL
LIN {X 0,Y 521.51,Z 303.398,A -85,B 0,C 180,E1 23718.393,E2 23718.393} C_VEL
LIN {X 0,Y 524.459,Z 316.445,A -85,B 0,C 180,E1 23717.109,E2 23717.109} C_VEL
LIN {X 0,Y 528.806,Z 327.323,A -85,B 0,C 180,E1 23715.909,E2 23715.909} C_VEL
LIN {X 0,Y 534.216,Z 336.078,A -85,B 0,C 180,E1 23714.818,E2 23714.818} C_VEL
LIN {X 0,Y 541.635,Z 344.237,A -85,B 0,C 180,E1 23713.662,E2 23713.662} C_VEL
LIN {X 0,Y 550.158,Z 350.606,A -85,B 0,C 180,E1 23712.605,E2 23712.605} C_VEL
LIN {X 0,Y 560.155,Z 355.601,A -85,B 0,C 180,E1 23711.591,E2 23711.591} C_VEL
LIN {X 0,Y 565.232,Z 357.247,A -85,B 0,C 180,E1 23711.1,E2 23711.1} C_VEL
LIN {X 0,Y 568.903,Z 357.611,A -85,B 0,C 180,E1 23710.602,E2 23710.602} C_VEL
LIN {X 0,Y 571.79,Z 356.876,A -85,B 0,C 180,E1 23710.013,E2 23710.013} C_VEL
LIN {X 0,Y 573.351,Z 355.116,A -85,B 0,C 180,E1 23709.403,E2 23709.403} C_VEL
LIN {X 0,Y 573.478,Z 352.298,A -85,B 0,C 180,E1 23708.785,E2 23708.785} C_VEL
LIN {X 0,Y 572.05,Z 348.682,A -85,B 0,C 180,E1 23708.224,E2 23708.224} C_VEL
LIN {X 0,Y 568.908,Z 344.107,A -85,B 0,C 180,E1 23707.722,E2 23707.722} C_VEL
LIN {X 0,Y 567.725,Z 342.723,A -85,B 0,C 180,E1 23707.567,E2 23707.567} C_VEL
LIN {X 0,Y 565.145,Z 354.806,A -85,B 0,C 180,E1 23707.226,E2 23707.226} C_VEL
LIN {X 0,Y 563.041,Z 374.27,A -85,B 0,C 180,E1 23707.049,E2 23707.049} C_VEL
LIN {X 0,Y 559.117,Z 392.818,A -85,B 0,C 180,E1 23706.942,E2 23706.942} C_VEL
LIN {X 0,Y 553.255,Z 411.126,A -85,B 0,C 180,E1 23706.841,E2 23706.841} C_VEL
LIN {X 0,Y 545.996,Z 428.453,A -85,B 0,C 180,E1 23706.67,E2 23706.67} C_VEL
LIN {X 0,Y 539.779,Z 442.249,A -85,B 0,C 180,E1 23706.352,E2 23706.352} C_VEL
LIN {X 0,Y 535.797,Z 451.853,A -85,B 0,C 180,E1 23706.003,E2 23706.003} C_VEL
LIN {X 0,Y 529.716,Z 463.991,A -85,B 0,C 180,E1 23705.679,E2 23705.679} C_VEL
LIN {X 0,Y 525.675,Z 473.866,A -85,B 0,C 180,E1 23705.259,E2 23705.259} C_VEL
LIN {X 0,Y 520.724,Z 487.028,A -85,B 0,C 180,E1 23704.636,E2 23704.636} C_VEL
LIN {X 0,Y 518.98,Z 493.055,A -85,B 0,C 180,E1 23704.332,E2 23704.332} C_VEL
LIN {X 0,Y 518.304,Z 534.254,A -85,B 0,C 180,E1 23703.659,E2 23703.659} C_VEL
LIN {X 0,Y 517.461,Z 556.486,A -85,B 0,C 180,E1 23703.096,E2 23703.096} C_VEL
LIN {X 0,Y 516.437,Z 578.065,A -85,B 0,C 180,E1 23702.333,E2 23702.333} C_VEL
LIN {X 0,Y 515.169,Z 599.522,A -85,B 0,C 180,E1 23701.355,E2 23701.355} C_VEL
LIN {X 0,Y 513.799,Z 619.764,A -85,B 0,C 180,E1 23700.202,E2 23700.202} C_VEL
LIN {X 0,Y 512.295,Z 639.782,A -85,B 0,C 180,E1 23698.821,E2 23698.821} C_VEL
LIN {X 0,Y 510.764,Z 659.493,A -85,B 0,C 180,E1 23697.2,E2 23697.2} C_VEL
LIN {X 0,Y 509.319,Z 677.597,A -85,B 0,C 180,E1 23695.44,E2 23695.44} C_VEL
LIN {X 0,Y 507.97,Z 694.819,A -85,B 0,C 180,E1 23693.474,E2 23693.474} C_VEL
LIN {X 0,Y 506.805,Z 710.473,A -85,B 0,C 180,E1 23691.379,E2 23691.379} C_VEL
LIN {X 0,Y 505.841,Z 724.806,A -85,B 0,C 180,E1 23689.122,E2 23689.122} C_VEL
LIN {X 0,Y 505.102,Z 737.287,A -85,B 0,C 180,E1 23686.799,E2 23686.799} C_VEL
LIN {X 0,Y 504.555,Z 748.505,A -85,B 0,C 180,E1 23684.297,E2 23684.297} C_VEL
LIN {X 0,Y 504.216,Z 757.701,A -85,B 0,C 180,E1 23681.785,E2 23681.785} C_VEL
LIN {X 0,Y 504.038,Z 765,A -85,B 0,C 180,E1 23679.246,E2 23679.246} C_VEL
LIN {X 0,Y 503.952,Z 770.225,A -85,B 0,C 180,E1 23676.837,E2 23676.837} C_VEL
LIN {X 0,Y 503.919,Z 773.874,A -85,B 0,C 180,E1 23674.438,E2 23674.438} C_VEL
LIN {X 0,Y 503.908,Z 775.975,A -85,B 0,C 180,E1 23671.933,E2 23671.933} C_VEL
LIN {X 0,Y 503.898,Z 776.431,A -85,B 0,C 180,E1 23669.431,E2 23669.431} C_VEL
LIN {X 0,Y 503.916,Z 775.231,A -85,B 0,C 180,E1 23666.929,E2 23666.929} C_VEL
LIN {X 0,Y 503.93,Z 772.339,A -85,B 0,C 180,E1 23664.421,E2 23664.421} C_VEL
LIN {X 0,Y 503.987,Z 767.633,A -85,B 0,C 180,E1 23661.875,E2 23661.875} C_VEL
LIN {X 0,Y 504.115,Z 761.264,A -85,B 0,C 180,E1 23659.37,E2 23659.37} C_VEL
LIN {X 0,Y 504.367,Z 753.267,A -85,B 0,C 180,E1 23656.938,E2 23656.938} C_VEL
LIN {X 0,Y 504.76,Z 743.845,A -85,B 0,C 180,E1 23654.607,E2 23654.607} C_VEL
LIN {X 0,Y 505.366,Z 732.488,A -85,B 0,C 180,E1 23652.26,E2 23652.26} C_VEL
LIN {X 0,Y 506.18,Z 719.628,A -85,B 0,C 180,E1 23650.018,E2 23650.018} C_VEL
LIN {X 0,Y 507.25,Z 704.353,A -85,B 0,C 180,E1 23647.762,E2 23647.762} C_VEL
LIN {X 0,Y 508.523,Z 687.705,A -85,B 0,C 180,E1 23645.674,E2 23645.674} C_VEL
LIN {X 0,Y 509.956,Z 669.74,A -85,B 0,C 180,E1 23643.76,E2 23643.76} C_VEL
LIN {X 0,Y 511.394,Z 651.345,A -85,B 0,C 180,E1 23642.096,E2 23642.096} C_VEL
LIN {X 0,Y 512.927,Z 631.501,A -85,B 0,C 180,E1 23640.578,E2 23640.578} C_VEL
LIN {X 0,Y 514.343,Z 611.752,A -85,B 0,C 180,E1 23639.317,E2 23639.317} C_VEL
LIN {X 0,Y 515.69,Z 591.178,A -85,B 0,C 180,E1 23638.237,E2 23638.237} C_VEL
LIN {X 0,Y 516.884,Z 569.488,A -85,B 0,C 180,E1 23637.337,E2 23637.337} C_VEL
LIN {X 0,Y 517.831,Z 548.089,A -85,B 0,C 180,E1 23636.666,E2 23636.666} C_VEL
LIN {X 0,Y 518.509,Z 525.81,A -85,B 0,C 180,E1 23636.181,E2 23636.181} C_VEL
LIN {X 0,Y 519.098,Z 490,A -85,B 0,C 180,E1 23635.608,E2 23635.608} C_VEL
LIN {X 0,Y 523.258,Z 471.043,A -85,B 0,C 180,E1 23634.889,E2 23634.889} C_VEL
LIN {X 0,Y 525.145,Z 463.598,A -85,B 0,C 180,E1 23634.633,E2 23634.633} C_VEL
LIN {X 0,Y 528.684,Z 449.915,A -85,B 0,C 180,E1 23634.173,E2 23634.173} C_VEL
LIN {X 0,Y 533.779,Z 434.188,A -85,B 0,C 180,E1 23633.773,E2 23633.773} C_VEL
LIN {X 0,Y 537.151,Z 421.161,A -85,B 0,C 180,E1 23633.347,E2 23633.347} C_VEL
LIN {X 0,Y 543.54,Z 401.642,A -85,B 0,C 180,E1 23632.921,E2 23632.921} C_VEL
LIN {X 0,Y 551.756,Z 377.469,A -85,B 0,C 180,E1 23632.622,E2 23632.622} C_VEL
LIN {X 0,Y 559.12,Z 352.496,A -85,B 0,C 180,E1 23632.442,E2 23632.442} C_VEL
LIN {X 0,Y 562.136,Z 340.482,A -85,B 0,C 180,E1 23632.11,E2 23632.11} C_VEL
LIN {X 0,Y 567.866,Z 316.814,A -85,B 0,C 180,E1 23631.758,E2 23631.758} C_VEL
LIN {X 0,Y 573.71,Z 286.809,A -85,B 0,C 180,E1 23631.465,E2 23631.465} C_VEL
LIN {X 0,Y 577.315,Z 259.415,A -85,B 0,C 180,E1 23631.206,E2 23631.206} C_VEL
LIN {X 0,Y 580.222,Z 261.999,A -85,B 0,C 180,E1 23630.643,E2 23630.643} C_VEL
LIN {X 0,Y 581.502,Z 263.848,A -85,B 0,C 180,E1 23630.049,E2 23630.049} C_VEL
LIN {X 0,Y 581.383,Z 264.97,A -85,B 0,C 180,E1 23629.452,E2 23629.452} C_VEL
LIN {X 0,Y 579.632,Z 265.437,A -85,B 0,C 180,E1 23628.772,E2 23628.772} C_VEL
LIN {X 0,Y 576.568,Z 265.516,A -85,B 0,C 180,E1 23628.218,E2 23628.218} C_VEL
LIN {X 0,Y 571.948,Z 264.476,A -85,B 0,C 180,E1 23627.686,E2 23627.686} C_VEL
LIN {X 0,Y 561.575,Z 260.078,A -85,B 0,C 180,E1 23626.736,E2 23626.736} C_VEL
LIN {X 0,Y 552.56,Z 254.208,A -85,B 0,C 180,E1 23625.771,E2 23625.771} C_VEL
LIN {X 0,Y 542.042,Z 245.776,A -85,B 0,C 180,E1 23624.503,E2 23624.503} C_VEL
LIN {X 0,Y 534.4,Z 236.739,A -85,B 0,C 180,E1 23623.365,E2 23623.365} C_VEL
LIN {X 0,Y 527.939,Z 224.9,A -85,B 0,C 180,E1 23622.1,E2 23622.1} C_VEL
LIN {X 0,Y 518.533,Z 205.009,A -85,B 0,C 180,E1 23619.949,E2 23619.949} C_VEL
LIN {X 0,Y 511.407,Z 191.773,A -85,B 0,C 180,E1 23618.299,E2 23618.299} C_VEL
LIN {X 0,Y 507.407,Z 184.116,A -85,B 0,C 180,E1 23617.296,E2 23617.296} C_VEL
LIN {X 0,Y 505.346,Z 181.217,A -85,B 0,C 180,E1 23616.834,E2 23616.834} C_VEL
LIN {X 0,Y 504.669,Z 178.872,A -85,B 0,C 180,E1 23616.567,E2 23616.567} C_VEL
LIN {X 0,Y 504.733,Z 179.026,A -85,B 0,C 180,E1 23613.511,E2 23613.511} C_VEL
LIN {X 0,Y 508.375,Z 191.505,A -85,B 0,C 180,E1 23612.462,E2 23612.462} C_VEL
LIN {X 0,Y 509.328,Z 226.327,A -85,B 0,C 180,E1 23609.909,E2 23609.909} C_VEL
LIN {X 0,Y 509.729,Z 254.47,A -85,B 0,C 180,E1 23607.703,E2 23607.703} C_VEL
LIN {X 0,Y 509.858,Z 285.446,A -85,B 0,C 180,E1 23605.185,E2 23605.185} C_VEL
LIN {X 0,Y 509.561,Z 321.318,A -85,B 0,C 180,E1 23602.132,E2 23602.132} C_VEL
LIN {X 0,Y 509.304,Z 326.504,A -85,B 0,C 180,E1 23601.727,E2 23601.727} C_VEL
LIN {X 0,Y 508.077,Z 459.701,A -85,B 0,C 180,E1 23599.696,E2 23599.696} C_VEL
LIN {X 0,Y 507.978,Z 494.607,A -85,B 0,C 180,E1 23599.157,E2 23599.157} C_VEL
LIN {X 0,Y 507.876,Z 512.039,A -85,B 0,C 180,E1 23598.665,E2 23598.665} C_VEL
LIN {X 0,Y 507.626,Z 528.8,A -85,B 0,C 180,E1 23597.976,E2 23597.976} C_VEL
LIN {X 0,Y 507.293,Z 544.096,A -85,B 0,C 180,E1 23597.137,E2 23597.137} C_VEL
LIN {X 0,Y 506.862,Z 558.904,A -85,B 0,C 180,E1 23596.09,E2 23596.09} C_VEL
LIN {X 0,Y 506.386,Z 572.652,A -85,B 0,C 180,E1 23594.873,E2 23594.873} C_VEL
LIN {X 0,Y 505.913,Z 585.336,A -85,B 0,C 180,E1 23593.486,E2 23593.486} C_VEL
LIN {X 0,Y 505.464,Z 596.403,A -85,B 0,C 180,E1 23591.987,E2 23591.987} C_VEL
LIN {X 0,Y 505.064,Z 606.399,A -85,B 0,C 180,E1 23590.295,E2 23590.295} C_VEL
LIN {X 0,Y 504.777,Z 614.602,A -85,B 0,C 180,E1 23588.543,E2 23588.543} C_VEL
LIN {X 0,Y 504.56,Z 621.185,A -85,B 0,C 180,E1 23586.714,E2 23586.714} C_VEL
LIN {X 0,Y 504.406,Z 626.168,A -85,B 0,C 180,E1 23584.775,E2 23584.775} C_VEL
LIN {X 0,Y 504.318,Z 629.525,A -85,B 0,C 180,E1 23582.727,E2 23582.727} C_VEL
LIN {X 0,Y 504.28,Z 630.979,A -85,B 0,C 180,E1 23580.795,E2 23580.795} C_VEL
LIN {X 0,Y 504.266,Z 630.687,A -85,B 0,C 180,E1 23578.75,E2 23578.75} C_VEL
LIN {X 0,Y 504.287,Z 628.589,A -85,B 0,C 180,E1 23576.699,E2 23576.699} C_VEL
LIN {X 0,Y 504.348,Z 624.893,A -85,B 0,C 180,E1 23574.767,E2 23574.767} C_VEL
LIN {X 0,Y 504.476,Z 619.3,A -85,B 0,C 180,E1 23572.827,E2 23572.827} C_VEL
LIN {X 0,Y 504.687,Z 612.183,A -85,B 0,C 180,E1 23570.995,E2 23570.995} C_VEL
LIN {X 0,Y 504.977,Z 603.618,A -85,B 0,C 180,E1 23569.273,E2 23569.273} C_VEL
LIN {X 0,Y 505.357,Z 593.573,A -85,B 0,C 180,E1 23567.661,E2 23567.661} C_VEL
LIN {X 0,Y 505.819,Z 582.029,A -85,B 0,C 180,E1 23566.161,E2 23566.161} C_VEL
LIN {X 0,Y 506.339,Z 568.927,A -85,B 0,C 180,E1 23564.773,E2 23564.773} C_VEL
LIN {X 0,Y 506.864,Z 554.739,A -85,B 0,C 180,E1 23563.556,E2 23563.556} C_VEL
LIN {X 0,Y 507.355,Z 539.594,A -85,B 0,C 180,E1 23562.523,E2 23562.523} C_VEL
LIN {X 0,Y 507.785,Z 522.872,A -85,B 0,C 180,E1 23561.636,E2 23561.636} C_VEL
LIN {X 0,Y 508.141,Z 505.863,A -85,B 0,C 180,E1 23560.97,E2 23560.97} C_VEL
LIN {X 0,Y 508.33,Z 488.144,A -85,B 0,C 180,E1 23560.509,E2 23560.509} C_VEL
LIN {X 0,Y 509.573,Z 324.536,A -85,B 0,C 180,E1 23558.017,E2 23558.017} C_VEL
LIN {X 0,Y 508.779,Z 319.649,A -85,B 0,C 180,E1 23557.893,E2 23557.893} C_VEL
LIN {X 0,Y 509.625,Z 281.414,A -85,B 0,C 180,E1 23554.366,E2 23554.366} C_VEL
LIN {X 0,Y 509.818,Z 269.499,A -85,B 0,C 180,E1 23553.264,E2 23553.264} C_VEL
LIN {X 0,Y 509.019,Z 263.778,A -85,B 0,C 180,E1 23552.683,E2 23552.683} C_VEL
LIN {X 0,Y 503.521,Z 249.386,A -85,B 0,C 180,E1 23551.023,E2 23551.023} C_VEL
LIN {X 0,Y 502.93,Z 244.405,A -85,B 0,C 180,E1 23550.521,E2 23550.521} C_VEL
LIN {X 0,Y 503.395,Z 208.782,A -85,B 0,C 180,E1 23547.231,E2 23547.231} C_VEL
LIN {X 0,Y 503.264,Z 200.745,A -85,B 0,C 180,E1 23546.473,E2 23546.473} C_VEL
LIN {X 0,Y 503.271,Z 200.578,A -85,B 0,C 180,E1 23546.423,E2 23546.423} C_VEL
LIN {X 0,Y 505.21,Z 202.324,A -85,B 0,C 180,E1 23546.211,E2 23546.211} C_VEL
LIN {X 0,Y 508.055,Z 202.402,A -85,B 0,C 180,E1 23545.949,E2 23545.949} C_VEL
LIN {X 0,Y 509.29,Z 202.184,A -85,B 0,C 180,E1 23545.841,E2 23545.841} C_VEL
LIN {X 0,Y 510.862,Z 202.746,A -85,B 0,C 180,E1 23545.689,E2 23545.689} C_VEL
LIN {X 0,Y 515.589,Z 210.679,A -85,B 0,C 180,E1 23545.135,E2 23545.135} C_VEL
LIN {X 0,Y 512.534,Z 405.843,A -85,B 0,C 180,E1 23542.046,E2 23542.046} C_VEL
LIN {X 0,Y 511.642,Z 464.339,A -85,B 0,C 180,E1 23541.109,E2 23541.109} C_VEL
LIN {X 0,Y 510.817,Z 484.889,A -85,B 0,C 180,E1 23540.59,E2 23540.59} C_VEL
LIN {X 0,Y 509.711,Z 506.129,A -85,B 0,C 180,E1 23539.85,E2 23539.85} C_VEL
LIN {X 0,Y 508.506,Z 525.5,A -85,B 0,C 180,E1 23538.984,E2 23538.984} C_VEL
LIN {X 0,Y 506.937,Z 547.037,A -85,B 0,C 180,E1 23537.784,E2 23537.784} C_VEL
LIN {X 0,Y 505.575,Z 564.394,A -85,B 0,C 180,E1 23536.619,E2 23536.619} C_VEL
LIN {X 0,Y 504.041,Z 582.904,A -85,B 0,C 180,E1 23535.168,E2 23535.168} C_VEL
LIN {X 0,Y 502.548,Z 599.777,A -85,B 0,C 180,E1 23533.596,E2 23533.596} C_VEL
LIN {X 0,Y 501.235,Z 614.915,A -85,B 0,C 180,E1 23531.984,E2 23531.984} C_VEL
LIN {X 0,Y 499.823,Z 631.789,A -85,B 0,C 180,E1 23529.893,E2 23529.893} C_VEL
LIN {X 0,Y 498.768,Z 644.989,A -85,B 0,C 180,E1 23527.983,E2 23527.983} C_VEL
LIN {X 0,Y 497.823,Z 658.308,A -85,B 0,C 180,E1 23525.764,E2 23525.764} C_VEL
LIN {X 0,Y 497.111,Z 669.367,A -85,B 0,C 180,E1 23523.582,E2 23523.582} C_VEL
LIN {X 0,Y 496.601,Z 679.247,A -85,B 0,C 180,E1 23521.296,E2 23521.296} C_VEL
LIN {X 0,Y 496.238,Z 688.124,A -85,B 0,C 180,E1 23518.779,E2 23518.779} C_VEL
LIN {X 0,Y 496.058,Z 694.365,A -85,B 0,C 180,E1 23516.581,E2 23516.581} C_VEL
LIN {X 0,Y 495.962,Z 700,A -85,B 0,C 180,E1 23514.031,E2 23514.031} C_VEL
LIN {X 0,Y 495.921,Z 703.607,A -85,B 0,C 180,E1 23511.649,E2 23511.649} C_VEL
LIN {X 0,Y 495.908,Z 705.74,A -85,B 0,C 180,E1 23509.309,E2 23509.309} C_VEL
LIN {X 0,Y 495.905,Z 706.444,A -85,B 0,C 180,E1 23506.637,E2 23506.637} C_VEL
LIN {X 0,Y 495.913,Z 705.571,A -85,B 0,C 180,E1 23504.359,E2 23504.359} C_VEL
LIN {X 0,Y 495.925,Z 703.142,A -85,B 0,C 180,E1 23501.868,E2 23501.868} C_VEL
LIN {X 0,Y 495.966,Z 698.821,A -85,B 0,C 180,E1 23499.281,E2 23499.281} C_VEL
LIN {X 0,Y 496.07,Z 693.682,A -85,B 0,C 180,E1 23497.063,E2 23497.063} C_VEL
LIN {X 0,Y 496.309,Z 686.529,A -85,B 0,C 180,E1 23494.622,E2 23494.622} C_VEL
LIN {X 0,Y 496.689,Z 677.519,A -85,B 0,C 180,E1 23492.192,E2 23492.192} C_VEL
LIN {X 0,Y 497.248,Z 667.295,A -85,B 0,C 180,E1 23489.885,E2 23489.885} C_VEL
LIN {X 0,Y 498.03,Z 655.091,A -85,B 0,C 180,E1 23487.584,E2 23487.584} C_VEL
LIN {X 0,Y 498.907,Z 643.077,A -85,B 0,C 180,E1 23485.633,E2 23485.633} C_VEL
LIN {X 0,Y 500.175,Z 627.568,A -85,B 0,C 180,E1 23483.457,E2 23483.457} C_VEL
LIN {X 0,Y 501.463,Z 612.277,A -85,B 0,C 180,E1 23481.631,E2 23481.631} C_VEL
LIN {X 0,Y 502.959,Z 595.332,A -85,B 0,C 180,E1 23479.867,E2 23479.867} C_VEL
LIN {X 0,Y 504.5,Z 577.233,A -85,B 0,C 180,E1 23478.279,E2 23478.279} C_VEL
LIN {X 0,Y 505.922,Z 560.06,A -85,B 0,C 180,E1 23476.98,E2 23476.98} C_VEL
LIN {X 0,Y 507.584,Z 538.648,A -85,B 0,C 180,E1 23475.629,E2 23475.629} C_VEL
LIN {X 0,Y 508.744,Z 521.421,A -85,B 0,C 180,E1 23474.731,E2 23474.731} C_VEL
LIN {X 0,Y 509.916,Z 502.476,A -85,B 0,C 180,E1 23473.917,E2 23473.917} C_VEL
LIN {X 0,Y 510.981,Z 481.431,A -85,B 0,C 180,E1 23473.221,E2 23473.221} C_VEL
LIN {X 0,Y 511.73,Z 460.183,A -85,B 0,C 180,E1 23472.72,E2 23472.72} C_VEL
LIN {X 0,Y 514.987,Z 252.986,A -85,B 0,C 180,E1 23469.426,E2 23469.426} C_VEL
LIN {X 0,Y 515.716,Z 210.24,A -85,B 0,C 180,E1 23468.725,E2 23468.725} C_VEL
LIN {X 0,Y 505.227,Z 193.735,A -85,B 0,C 180,E1 23467.443,E2 23467.443} C_VEL
LIN {X 0,Y 499.929,Z 185.471,A -85,B 0,C 180,E1 23466.764,E2 23466.764} C_VEL
LIN {X 0,Y 497.391,Z 182.139,A -85,B 0,C 180,E1 23466.443,E2 23466.443} C_VEL
LIN {X 0,Y 496.752,Z 179.857,A -85,B 0,C 180,E1 23466.324,E2 23466.324} C_VEL
LIN {X 0,Y 496.77,Z 179.854,A -85,B 0,C 180,E1 23462.814,E2 23462.814} C_VEL
LIN {X 0,Y 496.737,Z 179.859,A -85,B 0,C 180,E1 23459.386,E2 23459.386} C_VEL
LIN {X 0,Y 496.709,Z 179.858,A -85,B 0,C 180,E1 23455.826,E2 23455.826} C_VEL
LIN {X 0,Y 496.722,Z 179.852,A -85,B 0,C 180,E1 23452.271,E2 23452.271} C_VEL
LIN {X 0,Y 496.772,Z 179.845,A -85,B 0,C 180,E1 23448.83,E2 23448.83} C_VEL
LIN {X 0,Y 496.764,Z 179.846,A -85,B 0,C 180,E1 23445.214,E2 23445.214} C_VEL
LIN {X 0,Y 496.752,Z 179.851,A -85,B 0,C 180,E1 23441.623,E2 23441.623} C_VEL
LIN {X 0,Y 496.752,Z 179.856,A -85,B 0,C 180,E1 23438.094,E2 23438.094} C_VEL
LIN {X 0,Y 496.757,Z 179.858,A -85,B 0,C 180,E1 23434.584,E2 23434.584} C_VEL
LIN {X 0,Y 496.761,Z 179.85,A -85,B 0,C 180,E1 23430.97,E2 23430.97} C_VEL
LIN {X 0,Y 496.756,Z 179.847,A -85,B 0,C 180,E1 23427.423,E2 23427.423} C_VEL
LIN {X 0,Y 496.761,Z 179.853,A -85,B 0,C 180,E1 23423.864,E2 23423.864} C_VEL
LIN {X 0,Y 496.771,Z 179.856,A -85,B 0,C 180,E1 23420.255,E2 23420.255} C_VEL
LIN {X 0,Y 496.755,Z 179.852,A -85,B 0,C 180,E1 23416.728,E2 23416.728} C_VEL
LIN {X 0,Y 496.703,Z 179.85,A -85,B 0,C 180,E1 23413.385,E2 23413.385} C_VEL
LIN {X 0,Y 496.721,Z 179.856,A -85,B 0,C 180,E1 23409.852,E2 23409.852} C_VEL
LIN {X 0,Y 496.759,Z 179.855,A -85,B 0,C 180,E1 23406.356,E2 23406.356} C_VEL
LIN {X 0,Y 496.764,Z 179.854,A -85,B 0,C 180,E1 23402.769,E2 23402.769} C_VEL
LIN {X 0,Y 496.742,Z 179.854,A -85,B 0,C 180,E1 23399.193,E2 23399.193} C_VEL
LIN {X 0,Y 496.731,Z 179.85,A -85,B 0,C 180,E1 23395.729,E2 23395.729} C_VEL
LIN {X 0,Y 496.74,Z 179.85,A -85,B 0,C 180,E1 23392.25,E2 23392.25} C_VEL
LIN {X 0,Y 496.764,Z 179.849,A -85,B 0,C 180,E1 23388.742,E2 23388.742} C_VEL
LIN {X 0,Y 496.767,Z 179.85,A -85,B 0,C 180,E1 23385.19,E2 23385.19} C_VEL
LIN {X 0,Y 496.767,Z 179.849,A -85,B 0,C 180,E1 23381.579,E2 23381.579} C_VEL
LIN {X 0,Y 496.772,Z 179.849,A -85,B 0,C 180,E1 23378.015,E2 23378.015} C_VEL
LIN {X 0,Y 496.756,Z 179.86,A -85,B 0,C 180,E1 23374.486,E2 23374.486} C_VEL
LIN {X 0,Y 496.742,Z 180.009,A -85,B 0,C 180,E1 23371.863,E2 23371.863} C_VEL
LIN {X 0,Y 497.77,Z 182.968,A -85,B 0,C 180,E1 23371.441,E2 23371.441} C_VEL
LIN {X 0,Y 499.223,Z 185.496,A -85,B 0,C 180,E1 23371.009,E2 23371.009} C_VEL
LIN {X 0,Y 506.16,Z 199.484,A -85,B 0,C 180,E1 23368.832,E2 23368.832} C_VEL
LIN {X 0,Y 514.708,Z 217.439,A -85,B 0,C 180,E1 23366.245,E2 23366.245} C_VEL
LIN {X 0,Y 517.031,Z 222.871,A -85,B 0,C 180,E1 23365.519,E2 23365.519} C_VEL
LIN {X 0,Y 514.638,Z 263.917,A -85,B 0,C 180,E1 23362.254,E2 23362.254} C_VEL
LIN {X 0,Y 513.62,Z 291.863,A -85,B 0,C 180,E1 23360.029,E2 23360.029} C_VEL
LIN {X 0,Y 514.868,Z 307.043,A -85,B 0,C 180,E1 23358.68,E2 23358.68} C_VEL
LIN {X 0,Y 517.9,Z 320.512,A -85,B 0,C 180,E1 23357.341,E2 23357.341} C_VEL
LIN {X 0,Y 522.187,Z 331.454,A -85,B 0,C 180,E1 23356.121,E2 23356.121} C_VEL
LIN {X 0,Y 527.746,Z 340.703,A -85,B 0,C 180,E1 23354.965,E2 23354.965} C_VEL
LIN {X 0,Y 534.853,Z 348.856,A -85,B 0,C 180,E1 23353.814,E2 23353.814} C_VEL
LIN {X 0,Y 543.823,Z 355.94,A -85,B 0,C 180,E1 23352.657,E2 23352.657} C_VEL
LIN {X 0,Y 554.435,Z 361.544,A -85,B 0,C 180,E1 23351.548,E2 23351.548} C_VEL
LIN {X 0,Y 561.869,Z 364.132,A -85,B 0,C 180,E1 23350.862,E2 23350.862} C_VEL
LIN {X 0,Y 565.705,Z 364.605,A -85,B 0,C 180,E1 23350.38,E2 23350.38} C_VEL
LIN {X 0,Y 568.95,Z 363.948,A -85,B 0,C 180,E1 23349.768,E2 23349.768} C_VEL
LIN {X 0,Y 570.561,Z 362.534,A -85,B 0,C 180,E1 23349.235,E2 23349.235} C_VEL
LIN {X 0,Y 571.064,Z 359.841,A -85,B 0,C 180,E1 23348.59,E2 23348.59} C_VEL
LIN {X 0,Y 569.948,Z 356.371,A -85,B 0,C 180,E1 23348.007,E2 23348.007} C_VEL
LIN {X 0,Y 569.503,Z 355.825,A -85,B 0,C 180,E1 23347.898,E2 23347.898} C_VEL
LIN {X 0,Y 565.781,Z 373.854,A -85,B 0,C 180,E1 23347.823,E2 23347.823} C_VEL
LIN {X 0,Y 560.325,Z 391.073,A -85,B 0,C 180,E1 23347.768,E2 23347.768} C_VEL
LIN {X 0,Y 552.951,Z 408.328,A -85,B 0,C 180,E1 23347.675,E2 23347.675} C_VEL
LIN {X 0,Y 543.944,Z 425.425,A -85,B 0,C 180,E1 23347.476,E2 23347.476} C_VEL
LIN {X 0,Y 536.552,Z 438.993,A -85,B 0,C 180,E1 23347.14,E2 23347.14} C_VEL
LIN {X 0,Y 531.647,Z 449.572,A -85,B 0,C 180,E1 23346.731,E2 23346.731} C_VEL
LIN {X 0,Y 523.919,Z 463.124,A -85,B 0,C 180,E1 23346.271,E2 23346.271} C_VEL
LIN {X 0,Y 519.467,Z 473.167,A -85,B 0,C 180,E1 23345.812,E2 23345.812} C_VEL
LIN {X 0,Y 514.152,Z 486.708,A -85,B 0,C 180,E1 23345.143,E2 23345.143} C_VEL
LIN {X 0,Y 512.38,Z 492.846,A -85,B 0,C 180,E1 23344.841,E2 23344.841} C_VEL
LIN {X 0,Y 511.641,Z 533.927,A -85,B 0,C 180,E1 23344.162,E2 23344.162} C_VEL
LIN {X 0,Y 510.762,Z 556.107,A -85,B 0,C 180,E1 23343.599,E2 23343.599} C_VEL
LIN {X 0,Y 509.628,Z 577.983,A -85,B 0,C 180,E1 23342.822,E2 23342.822} C_VEL
LIN {X 0,Y 508.328,Z 598.536,A -85,B 0,C 180,E1 23341.879,E2 23341.879} C_VEL
LIN {X 0,Y 506.843,Z 618.823,A -85,B 0,C 180,E1 23340.726,E2 23340.726} C_VEL
LIN {X 0,Y 505.215,Z 638.991,A -85,B 0,C 180,E1 23339.329,E2 23339.329} C_VEL
LIN {X 0,Y 503.598,Z 657.915,A -85,B 0,C 180,E1 23337.769,E2 23337.769} C_VEL
LIN {X 0,Y 502.003,Z 676.275,A -85,B 0,C 180,E1 23335.988,E2 23335.988} C_VEL
LIN {X 0,Y 500.465,Z 694.221,A -85,B 0,C 180,E1 23333.926,E2 23333.926} C_VEL
LIN {X 0,Y 499.146,Z 710.292,A -85,B 0,C 180,E1 23331.751,E2 23331.751} C_VEL
LIN {X 0,Y 498.078,Z 724.619,A -85,B 0,C 180,E1 23329.465,E2 23329.465} C_VEL
LIN {X 0,Y 497.248,Z 737.291,A -85,B 0,C 180,E1 23327.072,E2 23327.072} C_VEL
LIN {X 0,Y 496.649,Z 748.332,A -85,B 0,C 180,E1 23324.575,E2 23324.575} C_VEL
LIN {X 0,Y 496.267,Z 757.31,A -85,B 0,C 180,E1 23322.095,E2 23322.095} C_VEL
LIN {X 0,Y 496.053,Z 764.405,A -85,B 0,C 180,E1 23319.631,E2 23319.631} C_VEL
LIN {X 0,Y 495.963,Z 769.806,A -85,B 0,C 180,E1 23317.18,E2 23317.18} C_VEL
LIN {X 0,Y 495.921,Z 773.741,A -85,B 0,C 180,E1 23314.626,E2 23314.626} C_VEL
LIN {X 0,Y 495.911,Z 775.91,A -85,B 0,C 180,E1 23312.08,E2 23312.08} C_VEL
LIN {X 0,Y 495.898,Z 776.447,A -85,B 0,C 180,E1 23309.538,E2 23309.538} C_VEL
LIN {X 0,Y 495.913,Z 775.424,A -85,B 0,C 180,E1 23307.111,E2 23307.111} C_VEL
LIN {X 0,Y 495.929,Z 772.658,A -85,B 0,C 180,E1 23304.562,E2 23304.562} C_VEL
LIN {X 0,Y 495.987,Z 768.201,A -85,B 0,C 180,E1 23302.004,E2 23302.004} C_VEL
LIN {X 0,Y 496.118,Z 762.245,A -85,B 0,C 180,E1 23299.549,E2 23299.549} C_VEL
LIN {X 0,Y 496.373,Z 754.521,A -85,B 0,C 180,E1 23297.08,E2 23297.08} C_VEL
LIN {X 0,Y 496.813,Z 744.827,A -85,B 0,C 180,E1 23294.58,E2 23294.58} C_VEL
LIN {X 0,Y 497.5,Z 733.123,A -85,B 0,C 180,E1 23292.091,E2 23292.091} C_VEL
LIN {X 0,Y 498.435,Z 719.628,A -85,B 0,C 180,E1 23289.694,E2 23289.694} C_VEL
LIN {X 0,Y 499.614,Z 704.354,A -85,B 0,C 180,E1 23287.403,E2 23287.403} C_VEL
LIN {X 0,Y 501.013,Z 687.708,A -85,B 0,C 180,E1 23285.285,E2 23285.285} C_VEL
LIN {X 0,Y 502.582,Z 669.745,A -85,B 0,C 180,E1 23283.345,E2 23283.345} C_VEL
LIN {X 0,Y 504.203,Z 650.897,A -85,B 0,C 180,E1 23281.622,E2 23281.622} C_VEL
LIN {X 0,Y 505.887,Z 630.641,A -85,B 0,C 180,E1 23280.062,E2 23280.062} C_VEL
LIN {X 0,Y 507.476,Z 610.425,A -85,B 0,C 180,E1 23278.769,E2 23278.769} C_VEL
LIN {X 0,Y 508.899,Z 589.908,A -85,B 0,C 180,E1 23277.696,E2 23277.696} C_VEL
LIN {X 0,Y 510.183,Z 568.153,A -85,B 0,C 180,E1 23276.801,E2 23276.801} C_VEL
LIN {X 0,Y 511.171,Z 546.734,A -85,B 0,C 180,E1 23276.136,E2 23276.136} C_VEL
LIN {X 0,Y 511.898,Z 523.157,A -85,B 0,C 180,E1 23275.642,E2 23275.642} C_VEL
LIN {X 0,Y 512.375,Z 490.151,A -85,B 0,C 180,E1 23275.126,E2 23275.126} C_VEL
LIN {X 0,Y 516.419,Z 471.577,A -85,B 0,C 180,E1 23274.422,E2 23274.422} C_VEL
LIN {X 0,Y 518.929,Z 461.666,A -85,B 0,C 180,E1 23274.069,E2 23274.069} C_VEL
LIN {X 0,Y 523.389,Z 446.104,A -85,B 0,C 180,E1 23273.55,E2 23273.55} C_VEL
LIN {X 0,Y 527.652,Z 434.33,A -85,B 0,C 180,E1 23273.216,E2 23273.216} C_VEL
LIN {X 0,Y 531.384,Z 420.537,A -85,B 0,C 180,E1 23272.755,E2 23272.755} C_VEL
LIN {X 0,Y 538.629,Z 400.796,A -85,B 0,C 180,E1 23272.259,E2 23272.259} C_VEL
LIN {X 0,Y 548.028,Z 377.629,A -85,B 0,C 180,E1 23271.88,E2 23271.88} C_VEL
LIN {X 0,Y 556.964,Z 354.084,A -85,B 0,C 180,E1 23271.666,E2 23271.666} C_VEL
LIN {X 0,Y 560.365,Z 341.559,A -85,B 0,C 180,E1 23271.321,E2 23271.321} C_VEL
LIN {X 0,Y 567.366,Z 318.097,A -85,B 0,C 180,E1 23270.961,E2 23270.961} C_VEL
LIN {X 0,Y 575.252,Z 288.482,A -85,B 0,C 180,E1 23270.696,E2 23270.696} C_VEL
LIN {X 0,Y 579.17,Z 270.496,A -85,B 0,C 180,E1 23270.557,E2 23270.557} C_VEL
LIN {X 0,Y 579.614,Z 272.121,A -85,B 0,C 180,E1 23269.886,E2 23269.886} C_VEL
LIN {X 0,Y 578.387,Z 272.876,A -85,B 0,C 180,E1 23269.215,E2 23269.215} C_VEL
LIN {X 0,Y 575.68,Z 273.052,A -85,B 0,C 180,E1 23268.617,E2 23268.617} C_VEL
LIN {X 0,Y 572.01,Z 272.597,A -85,B 0,C 180,E1 23268.128,E2 23268.128} C_VEL
LIN {X 0,Y 564.569,Z 270.202,A -85,B 0,C 180,E1 23267.454,E2 23267.454} C_VEL
LIN {X 0,Y 554.382,Z 265.187,A -85,B 0,C 180,E1 23266.471,E2 23266.471} C_VEL
LIN {X 0,Y 539.571,Z 254.287,A -85,B 0,C 180,E1 23264.762,E2 23264.762} C_VEL
LIN {X 0,Y 531.652,Z 246.01,A -85,B 0,C 180,E1 23263.646,E2 23263.646} C_VEL
LIN {X 0,Y 526.263,Z 238.022,A -85,B 0,C 180,E1 23262.708,E2 23262.708} C_VEL
LIN {X 0,Y 513.167,Z 210.611,A -85,B 0,C 180,E1 23259.723,E2 23259.723} C_VEL
LIN {X 0,Y 506.143,Z 197.378,A -85,B 0,C 180,E1 23258.049,E2 23258.049} C_VEL
LIN {X 0,Y 501.463,Z 188.93,A -85,B 0,C 180,E1 23256.881,E2 23256.881} C_VEL
LIN {X 0,Y 498.96,Z 184.468,A -85,B 0,C 180,E1 23256.238,E2 23256.238} C_VEL
LIN {X 0,Y 497.074,Z 181.278,A -85,B 0,C 180,E1 23255.756,E2 23255.756} C_VEL
LIN {X 0,Y 496.769,Z 179.844,A -85,B 0,C 180,E1 23255.568,E2 23255.568} C_VEL
LIN {X 0,Y 496.748,Z 179.865,A -85,B 0,C 180,E1 23253.933,E2 23253.933} C_VEL
LIN {X 0,Y 501.044,Z 193.62,A -85,B 0,C 180,E1 23252.737,E2 23252.737} C_VEL
LIN {X 0,Y 501.976,Z 228.425,A -85,B 0,C 180,E1 23250.178,E2 23250.178} C_VEL
LIN {X 0,Y 502.382,Z 257.615,A -85,B 0,C 180,E1 23247.885,E2 23247.885} C_VEL
LIN {X 0,Y 502.495,Z 288.222,A -85,B 0,C 180,E1 23245.395,E2 23245.395} C_VEL
LIN {X 0,Y 502.15,Z 325.352,A -85,B 0,C 180,E1 23242.229,E2 23242.229} C_VEL
LIN {X 0,Y 501.787,Z 328.549,A -85,B 0,C 180,E1 23242.013,E2 23242.013} C_VEL
LIN {X 0,Y 500.452,Z 454.133,A -85,B 0,C 180,E1 23240.039,E2 23240.039} C_VEL
LIN {X 0,Y 500.301,Z 495.893,A -85,B 0,C 180,E1 23239.388,E2 23239.388} C_VEL
LIN {X 0,Y 500.208,Z 513.216,A -85,B 0,C 180,E1 23238.897,E2 23238.897} C_VEL
LIN {X 0,Y 499.948,Z 530.492,A -85,B 0,C 180,E1 23238.179,E2 23238.179} C_VEL
LIN {X 0,Y 499.594,Z 546.29,A -85,B 0,C 180,E1 23237.295,E2 23237.295} C_VEL
LIN {X 0,Y 499.142,Z 561.058,A -85,B 0,C 180,E1 23236.226,E2 23236.226} C_VEL
LIN {X 0,Y 498.65,Z 574.735,A -85,B 0,C 180,E1 23234.99,E2 23234.99} C_VEL
LIN {X 0,Y 498.155,Z 587.351,A -85,B 0,C 180,E1 23233.581,E2 23233.581} C_VEL
LIN {X 0,Y 497.678,Z 598.31,A -85,B 0,C 180,E1 23232.06,E2 23232.06} C_VEL
LIN {X 0,Y 497.272,Z 607.808,A -85,B 0,C 180,E1 23230.425,E2 23230.425} C_VEL
LIN {X 0,Y 496.961,Z 615.895,A -85,B 0,C 180,E1 23228.678,E2 23228.678} C_VEL
LIN {X 0,Y 496.72,Z 622.526,A -85,B 0,C 180,E1 23226.82,E2 23226.82} C_VEL
LIN {X 0,Y 496.545,Z 627.53,A -85,B 0,C 180,E1 23224.851,E2 23224.851} C_VEL
LIN {X 0,Y 496.443,Z 630.888,A -85,B 0,C 180,E1 23222.77,E2 23222.77} C_VEL
LIN {X 0,Y 496.396,Z 632.331,A -85,B 0,C 180,E1 23220.807,E2 23220.807} C_VEL
LIN {X 0,Y 496.378,Z 632.078,A -85,B 0,C 180,E1 23218.845,E2 23218.845} C_VEL
LIN {X 0,Y 496.394,Z 630.036,A -85,B 0,C 180,E1 23216.766,E2 23216.766} C_VEL
LIN {X 0,Y 496.461,Z 626.379,A -85,B 0,C 180,E1 23214.8,E2 23214.8} C_VEL
LIN {X 0,Y 496.6,Z 620.847,A -85,B 0,C 180,E1 23212.829,E2 23212.829} C_VEL
LIN {X 0,Y 496.843,Z 613.272,A -85,B 0,C 180,E1 23210.852,E2 23210.852} C_VEL
LIN {X 0,Y 497.16,Z 604.617,A -85,B 0,C 180,E1 23209.102,E2 23209.102} C_VEL
LIN {X 0,Y 497.571,Z 594.459,A -85,B 0,C 180,E1 23207.465,E2 23207.465} C_VEL
LIN {X 0,Y 498.091,Z 582.312,A -85,B 0,C 180,E1 23205.883,E2 23205.883} C_VEL
LIN {X 0,Y 498.625,Z 569.572,A -85,B 0,C 180,E1 23204.532,E2 23204.532} C_VEL
LIN {X 0,Y 499.179,Z 555.184,A -85,B 0,C 180,E1 23203.295,E2 23203.295} C_VEL
LIN {X 0,Y 499.709,Z 539.618,A -85,B 0,C 180,E1 23202.233,E2 23202.233} C_VEL
LIN {X 0,Y 500.146,Z 523.336,A -85,B 0,C 180,E1 23201.369,E2 23201.369} C_VEL
LIN {X 0,Y 500.505,Z 506.284,A -85,B 0,C 180,E1 23200.703,E2 23200.703} C_VEL
LIN {X 0,Y 500.695,Z 488.543,A -85,B 0,C 180,E1 23200.242,E2 23200.242} C_VEL
LIN {X 0,Y 502.057,Z 325.476,A -85,B 0,C 180,E1 23197.711,E2 23197.711} C_VEL
LIN {X 0,Y 501.273,Z 320.518,A -85,B 0,C 180,E1 23197.574,E2 23197.574} C_VEL
LIN {X 0,Y 502.154,Z 283.179,A -85,B 0,C 180,E1 23194.112,E2 23194.112} C_VEL
LIN {X 0,Y 502.896,Z 245.83,A -85,B 0,C 180,E1 23190.653,E2 23190.653} C_VEL
LIN {X 0,Y 502.93,Z 244.405,A -85,B 0,C 180,E1 23190.521,E2 23190.521} C_VEL
LIN {X 0,Y 502.115,Z 238.678,A -85,B 0,C 180,E1 23189.935,E2 23189.935} C_VEL
LIN {X 0,Y 496.564,Z 224.319,A -85,B 0,C 180,E1 23188.253,E2 23188.253} C_VEL
LIN {X 0,Y 495.924,Z 219.277,A -85,B 0,C 180,E1 23187.745,E2 23187.745} C_VEL
LIN {X 0,Y 496.125,Z 210.655,A -85,B 0,C 180,E1 23186.913,E2 23186.913} C_VEL
LIN {X 0,Y 497.657,Z 212.3,A -85,B 0,C 180,E1 23186.736,E2 23186.736} C_VEL
LIN {X 0,Y 500.06,Z 212.476,A -85,B 0,C 180,E1 23186.505,E2 23186.505} C_VEL
LIN {X 0,Y 503.512,Z 210.525,A -85,B 0,C 180,E1 23186.219,E2 23186.219} C_VEL
LIN {X 0,Y 504.655,Z 210.44,A -85,B 0,C 180,E1 23186.115,E2 23186.115} C_VEL
LIN {X 0,Y 507.345,Z 210.615,A -85,B 0,C 180,E1 23185.866,E2 23185.866} C_VEL
LIN {X 0,Y 509.225,Z 214.022,A -85,B 0,C 180,E1 23185.636,E2 23185.636} C_VEL
LIN {X 0,Y 505.585,Z 421.155,A -85,B 0,C 180,E1 23182.297,E2 23182.297} C_VEL
LIN {X 0,Y 504.802,Z 466.432,A -85,B 0,C 180,E1 23181.549,E2 23181.549} C_VEL
LIN {X 0,Y 503.902,Z 488.141,A -85,B 0,C 180,E1 23180.986,E2 23180.986} C_VEL
LIN {X 0,Y 502.766,Z 508.905,A -85,B 0,C 180,E1 23180.232,E2 23180.232} C_VEL
LIN {X 0,Y 501.379,Z 529.566,A -85,B 0,C 180,E1 23179.271,E2 23179.271} C_VEL
LIN {X 0,Y 499.837,Z 548.46,A -85,B 0,C 180,E1 23178.172,E2 23178.172} C_VEL
LIN {X 0,Y 498.461,Z 564.615,A -85,B 0,C 180,E1 23177.067,E2 23177.067} C_VEL
LIN {X 0,Y 496.735,Z 583.804,A -85,B 0,C 180,E1 23175.534,E2 23175.534} C_VEL
LIN {X 0,Y 495.108,Z 600.757,A -85,B 0,C 180,E1 23173.923,E2 23173.923} C_VEL
LIN {X 0,Y 493.671,Z 616.088,A -85,B 0,C 180,E1 23172.254,E2 23172.254} C_VEL
LIN {X 0,Y 492.184,Z 632.292,A -85,B 0,C 180,E1 23170.196,E2 23170.196} C_VEL
LIN {X 0,Y 491.026,Z 645.524,A -85,B 0,C 180,E1 23168.245,E2 23168.245} C_VEL
LIN {X 0,Y 489.943,Z 659.48,A -85,B 0,C 180,E1 23165.853,E2 23165.853} C_VEL
LIN {X 0,Y 489.183,Z 670.373,A -85,B 0,C 180,E1 23163.636,E2 23163.636} C_VEL
LIN {X 0,Y 488.616,Z 680.611,A -85,B 0,C 180,E1 23161.179,E2 23161.179} C_VEL
LIN {X 0,Y 488.254,Z 688.75,A -85,B 0,C 180,E1 23158.767,E2 23158.767} C_VEL
LIN {X 0,Y 488.065,Z 694.907,A -85,B 0,C 180,E1 23156.526,E2 23156.526} C_VEL
LIN {X 0,Y 487.962,Z 700.371,A -85,B 0,C 180,E1 23153.936,E2 23153.936} C_VEL
LIN {X 0,Y 487.922,Z 703.85,A -85,B 0,C 180,E1 23151.51,E2 23151.51} C_VEL
LIN {X 0,Y 487.911,Z 705.869,A -85,B 0,C 180,E1 23149.14,E2 23149.14} C_VEL
LIN {X 0,Y 487.905,Z 706.405,A -85,B 0,C 180,E1 23146.428,E2 23146.428} C_VEL
LIN {X 0,Y 487.917,Z 705.431,A -85,B 0,C 180,E1 23144.115,E2 23144.115} C_VEL
LIN {X 0,Y 487.927,Z 702.878,A -85,B 0,C 180,E1 23141.585,E2 23141.585} C_VEL
LIN {X 0,Y 487.984,Z 698.561,A -85,B 0,C 180,E1 23139.03,E2 23139.03} C_VEL
LIN {X 0,Y 488.102,Z 693.489,A -85,B 0,C 180,E1 23136.824,E2 23136.824} C_VEL
LIN {X 0,Y 488.377,Z 685.881,A -85,B 0,C 180,E1 23134.227,E2 23134.227} C_VEL
LIN {X 0,Y 488.787,Z 677.225,A -85,B 0,C 180,E1 23131.876,E2 23131.876} C_VEL
LIN {X 0,Y 489.416,Z 666.962,A -85,B 0,C 180,E1 23129.532,E2 23129.532} C_VEL
LIN {X 0,Y 490.29,Z 654.689,A -85,B 0,C 180,E1 23127.195,E2 23127.195} C_VEL
LIN {X 0,Y 491.264,Z 642.633,A -85,B 0,C 180,E1 23125.213,E2 23125.213} C_VEL
LIN {X 0,Y 492.652,Z 627.02,A -85,B 0,C 180,E1 23123.006,E2 23123.006} C_VEL
LIN {X 0,Y 494.033,Z 612.174,A -85,B 0,C 180,E1 23121.211,E2 23121.211} C_VEL
LIN {X 0,Y 495.667,Z 595.209,A -85,B 0,C 180,E1 23119.423,E2 23119.423} C_VEL
LIN {X 0,Y 497.331,Z 577.074,A -85,B 0,C 180,E1 23117.813,E2 23117.813} C_VEL
LIN {X 0,Y 498.884,Z 559.862,A -85,B 0,C 180,E1 23116.498,E2 23116.498} C_VEL
LIN {X 0,Y 500.636,Z 538.889,A -85,B 0,C 180,E1 23115.159,E2 23115.159} C_VEL
LIN {X 0,Y 501.934,Z 521.145,A -85,B 0,C 180,E1 23114.222,E2 23114.222} C_VEL
LIN {X 0,Y 503.308,Z 500.751,A -85,B 0,C 180,E1 23113.348,E2 23113.348} C_VEL
LIN {X 0,Y 504.348,Z 479.632,A -85,B 0,C 180,E1 23112.671,E2 23112.671} C_VEL
LIN {X 0,Y 505.071,Z 457.598,A -85,B 0,C 180,E1 23112.179,E2 23112.179} C_VEL
LIN {X 0,Y 508.567,Z 260.175,A -85,B 0,C 180,E1 23108.985,E2 23108.985} C_VEL
LIN {X 0,Y 509.365,Z 213.412,A -85,B 0,C 180,E1 23108.2,E2 23108.2} C_VEL
LIN {X 0,Y 500.016,Z 198.725,A -85,B 0,C 180,E1 23107.025,E2 23107.025} C_VEL
LIN {X 0,Y 494.061,Z 189.901,A -85,B 0,C 180,E1 23106.251,E2 23106.251} C_VEL
LIN {X 0,Y 491.324,Z 185.724,A -85,B 0,C 180,E1 23105.884,E2 23105.884} C_VEL
LIN {X 0,Y 489.296,Z 182.718,A -85,B 0,C 180,E1 23105.611,E2 23105.611} C_VEL
LIN {X 0,Y 488.827,Z 180.845,A -85,B 0,C 180,E1 23105.502,E2 23105.502} C_VEL
LIN {X 0,Y 488.823,Z 180.844,A -85,B 0,C 180,E1 23101.937,E2 23101.937} C_VEL
LIN {X 0,Y 488.825,Z 180.837,A -85,B 0,C 180,E1 23098.424,E2 23098.424} C_VEL
LIN {X 0,Y 488.809,Z 180.838,A -85,B 0,C 180,E1 23094.906,E2 23094.906} C_VEL
LIN {X 0,Y 488.797,Z 180.839,A -85,B 0,C 180,E1 23091.39,E2 23091.39} C_VEL
LIN {X 0,Y 488.803,Z 180.837,A -85,B 0,C 180,E1 23087.861,E2 23087.861} C_VEL
LIN {X 0,Y 488.819,Z 180.833,A -85,B 0,C 180,E1 23084.227,E2 23084.227} C_VEL
LIN {X 0,Y 488.836,Z 180.831,A -85,B 0,C 180,E1 23080.638,E2 23080.638} C_VEL
LIN {X 0,Y 488.797,Z 180.842,A -85,B 0,C 180,E1 23077.117,E2 23077.117} C_VEL
LIN {X 0,Y 488.766,Z 180.85,A -85,B 0,C 180,E1 23073.634,E2 23073.634} C_VEL
LIN {X 0,Y 488.789,Z 180.848,A -85,B 0,C 180,E1 23070.078,E2 23070.078} C_VEL
LIN {X 0,Y 488.827,Z 180.839,A -85,B 0,C 180,E1 23066.613,E2 23066.613} C_VEL
LIN {X 0,Y 488.821,Z 180.83,A -85,B 0,C 180,E1 23063.008,E2 23063.008} C_VEL
LIN {X 0,Y 488.804,Z 180.842,A -85,B 0,C 180,E1 23059.441,E2 23059.441} C_VEL
LIN {X 0,Y 488.794,Z 180.85,A -85,B 0,C 180,E1 23055.909,E2 23055.909} C_VEL
LIN {X 0,Y 488.805,Z 180.841,A -85,B 0,C 180,E1 23052.403,E2 23052.403} C_VEL
LIN {X 0,Y 488.83,Z 180.833,A -85,B 0,C 180,E1 23048.825,E2 23048.825} C_VEL
LIN {X 0,Y 488.826,Z 180.839,A -85,B 0,C 180,E1 23045.282,E2 23045.282} C_VEL
LIN {X 0,Y 488.828,Z 180.846,A -85,B 0,C 180,E1 23041.641,E2 23041.641} C_VEL
LIN {X 0,Y 488.832,Z 180.844,A -85,B 0,C 180,E1 23038.125,E2 23038.125} C_VEL
LIN {X 0,Y 488.821,Z 180.842,A -85,B 0,C 180,E1 23034.484,E2 23034.484} C_VEL
LIN {X 0,Y 488.789,Z 180.843,A -85,B 0,C 180,E1 23030.938,E2 23030.938} C_VEL
LIN {X 0,Y 488.797,Z 180.841,A -85,B 0,C 180,E1 23027.478,E2 23027.478} C_VEL
LIN {X 0,Y 488.813,Z 180.843,A -85,B 0,C 180,E1 23023.848,E2 23023.848} C_VEL
LIN {X 0,Y 488.831,Z 180.844,A -85,B 0,C 180,E1 23020.276,E2 23020.276} C_VEL
LIN {X 0,Y 488.804,Z 180.847,A -85,B 0,C 180,E1 23016.748,E2 23016.748} C_VEL
LIN {X 0,Y 488.768,Z 180.843,A -85,B 0,C 180,E1 23013.254,E2 23013.254} C_VEL
LIN {X 0,Y 488.796,Z 180.965,A -85,B 0,C 180,E1 23012.831,E2 23012.831} C_VEL
LIN {X 0,Y 490.208,Z 184.448,A -85,B 0,C 180,E1 23012.287,E2 23012.287} C_VEL
LIN {X 0,Y 491.248,Z 186.383,A -85,B 0,C 180,E1 23011.955,E2 23011.955} C_VEL
LIN {X 0,Y 497.776,Z 199.351,A -85,B 0,C 180,E1 23009.857,E2 23009.857} C_VEL
LIN {X 0,Y 506.902,Z 218.424,A -85,B 0,C 180,E1 23007.016,E2 23007.016} C_VEL
LIN {X 0,Y 510.578,Z 226.729,A -85,B 0,C 180,E1 23005.872,E2 23005.872} C_VEL
LIN {X 0,Y 508.029,Z 267.21,A -85,B 0,C 180,E1 23002.623,E2 23002.623} C_VEL
LIN {X 0,Y 506.948,Z 294.487,A -85,B 0,C 180,E1 23000.428,E2 23000.428} C_VEL
LIN {X 0,Y 508.197,Z 310.457,A -85,B 0,C 180,E1 22998.994,E2 22998.994} C_VEL
LIN {X 0,Y 511.155,Z 323.988,A -85,B 0,C 180,E1 22997.634,E2 22997.634} C_VEL
LIN {X 0,Y 515.618,Z 335.664,A -85,B 0,C 180,E1 22996.328,E2 22996.328} C_VEL
LIN {X 0,Y 521.331,Z 345.386,A -85,B 0,C 180,E1 22995.107,E2 22995.107} C_VEL
LIN {X 0,Y 528.622,Z 353.965,A -85,B 0,C 180,E1 22993.893,E2 22993.893} C_VEL
LIN {X 0,Y 537.505,Z 361.23,A -85,B 0,C 180,E1 22992.712,E2 22992.712} C_VEL
LIN {X 0,Y 547.997,Z 367.124,A -85,B 0,C 180,E1 22991.577,E2 22991.577} C_VEL
LIN {X 0,Y 558.494,Z 370.995,A -85,B 0,C 180,E1 22990.617,E2 22990.617} C_VEL
LIN {X 0,Y 563.091,Z 371.577,A -85,B 0,C 180,E1 22990.066,E2 22990.066} C_VEL
LIN {X 0,Y 566.359,Z 370.896,A -85,B 0,C 180,E1 22989.461,E2 22989.461} C_VEL
LIN {X 0,Y 568.027,Z 369.455,A -85,B 0,C 180,E1 22988.921,E2 22988.921} C_VEL
LIN {X 0,Y 568.459,Z 368.424,A -85,B 0,C 180,E1 22988.639,E2 22988.639} C_VEL
LIN {X 0,Y 561.643,Z 385.293,A -85,B 0,C 180,E1 22988.6,E2 22988.6} C_VEL
LIN {X 0,Y 553.159,Z 401.651,A -85,B 0,C 180,E1 22988.495,E2 22988.495} C_VEL
LIN {X 0,Y 542.624,Z 418.574,A -85,B 0,C 180,E1 22988.252,E2 22988.252} C_VEL
LIN {X 0,Y 533.418,Z 432.749,A -85,B 0,C 180,E1 22987.864,E2 22987.864} C_VEL
LIN {X 0,Y 526.806,Z 444.836,A -85,B 0,C 180,E1 22987.398,E2 22987.398} C_VEL
LIN {X 0,Y 524.385,Z 449.787,A -85,B 0,C 180,E1 22987.188,E2 22987.188} C_VEL
LIN {X 0,Y 517.288,Z 461.781,A -85,B 0,C 180,E1 22986.743,E2 22986.743} C_VEL
LIN {X 0,Y 512.473,Z 472.638,A -85,B 0,C 180,E1 22986.24,E2 22986.24} C_VEL
LIN {X 0,Y 507.113,Z 486.185,A -85,B 0,C 180,E1 22985.566,E2 22985.566} C_VEL
LIN {X 0,Y 505.994,Z 490.014,A -85,B 0,C 180,E1 22985.394,E2 22985.394} C_VEL
LIN {X 0,Y 505.042,Z 531.176,A -85,B 0,C 180,E1 22984.719,E2 22984.719} C_VEL
LIN {X 0,Y 504.033,Z 554.38,A -85,B 0,C 180,E1 22984.131,E2 22984.131} C_VEL
LIN {X 0,Y 502.827,Z 576.23,A -85,B 0,C 180,E1 22983.368,E2 22983.368} C_VEL
LIN {X 0,Y 501.527,Z 597.156,A -85,B 0,C 180,E1 22982.431,E2 22982.431} C_VEL
LIN {X 0,Y 500.007,Z 616.82,A -85,B 0,C 180,E1 22981.327,E2 22981.327} C_VEL
LIN {X 0,Y 498.327,Z 636.611,A -85,B 0,C 180,E1 22979.973,E2 22979.973} C_VEL
LIN {X 0,Y 496.595,Z 655.211,A -85,B 0,C 180,E1 22978.456,E2 22978.456} C_VEL
LIN {X 0,Y 494.842,Z 673.915,A -85,B 0,C 180,E1 22976.652,E2 22976.652} C_VEL
LIN {X 0,Y 493.25,Z 690.685,A -85,B 0,C 180,E1 22974.752,E2 22974.752} C_VEL
LIN {X 0,Y 491.843,Z 706.063,A -85,B 0,C 180,E1 22972.721,E2 22972.721} C_VEL
LIN {X 0,Y 490.647,Z 720.35,A -85,B 0,C 180,E1 22970.518,E2 22970.518} C_VEL
LIN {X 0,Y 489.637,Z 733.74,A -85,B 0,C 180,E1 22968.083,E2 22968.083} C_VEL
LIN {X 0,Y 488.888,Z 745.41,A -85,B 0,C 180,E1 22965.54,E2 22965.54} C_VEL
LIN {X 0,Y 488.407,Z 755.053,A -85,B 0,C 180,E1 22962.978,E2 22962.978} C_VEL
LIN {X 0,Y 488.125,Z 762.895,A -85,B 0,C 180,E1 22960.385,E2 22960.385} C_VEL
LIN {X 0,Y 487.979,Z 768.917,A -85,B 0,C 180,E1 22957.772,E2 22957.772} C_VEL
LIN {X 0,Y 487.928,Z 772.978,A -85,B 0,C 180,E1 22955.291,E2 22955.291} C_VEL
LIN {X 0,Y 487.91,Z 775.571,A -85,B 0,C 180,E1 22952.701,E2 22952.701} C_VEL
LIN {X 0,Y 487.91,Z 776.489,A -85,B 0,C 180,E1 22950.117,E2 22950.117} C_VEL
LIN {X 0,Y 487.91,Z 775.778,A -85,B 0,C 180,E1 22947.651,E2 22947.651} C_VEL
LIN {X 0,Y 487.924,Z 773.588,A -85,B 0,C 180,E1 22945.18,E2 22945.18} C_VEL
LIN {X 0,Y 487.965,Z 769.597,A -85,B 0,C 180,E1 22942.583,E2 22942.583} C_VEL
LIN {X 0,Y 488.087,Z 763.806,A -85,B 0,C 180,E1 22939.972,E2 22939.972} C_VEL
LIN {X 0,Y 488.348,Z 756.527,A -85,B 0,C 180,E1 22937.465,E2 22937.465} C_VEL
